LIN {X 0,Y 572.99,Z 934.788,A -85,B 0,C 180,E1 -2246.836,E2 -2246.836} C_VEL
LIN {X 0,Y 572.937,Z 937.681,A -85,B 0,C 180,E1 -2247.891,E2 -2247.891} C_VEL
LIN {X 0,Y 572.945,Z 938.936,A -85,B 0,C 180,E1 -2248.594,E2 -2248.594} C_VEL
LIN {X 0,Y 572.938,Z 939.711,A -85,B 0,C 180,E1 -2249.297,E2 -2249.297} C_VEL
LIN {X 0,Y 572.935,Z 940,A -85,B 0,C 180,E1 -2250,E2 -2250} C_VEL
LIN {X 0,Y 572.938,Z 939.711,A -85,B 0,C 180,E1 -2250.703,E2 -2250.703} C_VEL
LIN {X 0,Y 572.945,Z 938.936,A -85,B 0,C 180,E1 -2251.406,E2 -2251.406} C_VEL
LIN {X 0,Y 572.937,Z 937.68,A -85,B 0,C 180,E1 -2252.109,E2 -2252.109} C_VEL
LIN {X 0,Y 572.99,Z 934.788,A -85,B 0,C 180,E1 -2253.164,E2 -2253.164} C_VEL
LIN {X 0,Y 573.036,Z 932.147,A -85,B 0,C 180,E1 -2253.868,E2 -2253.868} C_VEL
LIN {X 0,Y 572.995,Z 926.985,A -85,B 0,C 180,E1 -2254.925,E2 -2254.925} C_VEL
LIN {X 0,Y 573.137,Z 920.188,A -85,B 0,C 180,E1 -2255.983,E2 -2255.983} C_VEL
LIN {X 0,Y 573.164,Z 912.803,A -85,B 0,C 180,E1 -2256.86,E2 -2256.86} C_VEL
LIN {X 0,Y 573.216,Z 905.405,A -85,B 0,C 180,E1 -2257.574,E2 -2257.574} C_VEL
LIN {X 0,Y 573.284,Z 897.548,A -85,B 0,C 180,E1 -2258.193,E2 -2258.193} C_VEL
LIN {X 0,Y 573.4,Z 887.734,A -85,B 0,C 180,E1 -2258.813,E2 -2258.813} C_VEL
LIN {X 0,Y 573.443,Z 876.299,A -85,B 0,C 180,E1 -2259.346,E2 -2259.346} C_VEL
LIN {X 0,Y 573.53,Z 866.245,A -85,B 0,C 180,E1 -2259.678,E2 -2259.678} C_VEL
LIN {X 0,Y 573.574,Z 857.443,A -85,B 0,C 180,E1 -2259.877,E2 -2259.877} C_VEL
LIN {X 0,Y 573.574,Z 783.105,A -85,B 0,C 180,E1 -2260.826,E2 -2260.826} C_VEL
LIN {X 0,Y 573.197,Z 780.107,A -85,B 0,C 180,E1 -2260.899,E2 -2260.899} C_VEL
LIN {X 0,Y 573.231,Z 774.077,A -85,B 0,C 180,E1 -2261.851,E2 -2261.851} C_VEL
LIN {X 0,Y 573.374,Z 755.693,A -85,B 0,C 180,E1 -2264.916,E2 -2264.916} C_VEL
LIN {X 0,Y 573.523,Z 738.39,A -85,B 0,C 180,E1 -2267.84,E2 -2267.84} C_VEL
LIN {X 0,Y 573.707,Z 721.087,A -85,B 0,C 180,E1 -2270.809,E2 -2270.809} C_VEL
LIN {X 0,Y 573.325,Z 716.043,A -85,B 0,C 180,E1 -2271.719,E2 -2271.719} C_VEL
LIN {X 0,Y 573.27,Z 715.887,A -85,B 0,C 180,E1 -2274.879,E2 -2274.879} C_VEL
LIN {X 0,Y 573.273,Z 715.885,A -85,B 0,C 180,E1 -2277.766,E2 -2277.766} C_VEL
LIN {X 0,Y 573.251,Z 715.882,A -85,B 0,C 180,E1 -2280.176,E2 -2280.176} C_VEL
LIN {X 0,Y 573.257,Z 715.884,A -85,B 0,C 180,E1 -2282.645,E2 -2282.645} C_VEL
LIN {X 0,Y 573.271,Z 715.889,A -85,B 0,C 180,E1 -2285.183,E2 -2285.183} C_VEL
LIN {X 0,Y 573.238,Z 715.891,A -85,B 0,C 180,E1 -2287.807,E2 -2287.807} C_VEL
LIN {X 0,Y 573.271,Z 715.88,A -85,B 0,C 180,E1 -2290.528,E2 -2290.528} C_VEL
LIN {X 0,Y 573.245,Z 715.894,A -85,B 0,C 180,E1 -2293.669,E2 -2293.669} C_VEL
LIN {X 0,Y 573.242,Z 715.885,A -85,B 0,C 180,E1 -2296.641,E2 -2296.641} C_VEL
LIN {X 0,Y 573.276,Z 715.885,A -85,B 0,C 180,E1 -2299.478,E2 -2299.478} C_VEL
LIN {X 0,Y 573.239,Z 715.886,A -85,B 0,C 180,E1 -2302.193,E2 -2302.193} C_VEL
LIN {X 0,Y 573.271,Z 715.881,A -85,B 0,C 180,E1 -2304.817,E2 -2304.817} C_VEL
LIN {X 0,Y 573.257,Z 715.887,A -85,B 0,C 180,E1 -2307.355,E2 -2307.355} C_VEL
LIN {X 0,Y 573.252,Z 715.893,A -85,B 0,C 180,E1 -2309.824,E2 -2309.824} C_VEL
LIN {X 0,Y 573.275,Z 715.887,A -85,B 0,C 180,E1 -2312.234,E2 -2312.234} C_VEL
LIN {X 0,Y 573.269,Z 715.882,A -85,B 0,C 180,E1 -2315.122,E2 -2315.122} C_VEL
LIN {X 0,Y 573.239,Z 715.889,A -85,B 0,C 180,E1 -2317.662,E2 -2317.662} C_VEL
LIN {X 0,Y 573.281,Z 715.882,A -85,B 0,C 180,E1 -2320.728,E2 -2320.728} C_VEL
LIN {X 0,Y 573.255,Z 715.886,A -85,B 0,C 180,E1 -2323.622,E2 -2323.622} C_VEL
LIN {X 0,Y 573.276,Z 715.884,A -85,B 0,C 180,E1 -2325.807,E2 -2325.807} C_VEL
LIN {X 0,Y 573.265,Z 715.884,A -85,B 0,C 180,E1 -2328.745,E2 -2328.745} C_VEL
LIN {X 0,Y 573.292,Z 715.88,A -85,B 0,C 180,E1 -2331.541,E2 -2331.541} C_VEL
LIN {X 0,Y 573.288,Z 715.89,A -85,B 0,C 180,E1 -2334.372,E2 -2334.372} C_VEL
LIN {X 0,Y 573.312,Z 715.875,A -85,B 0,C 180,E1 -2337.893,E2 -2337.893} C_VEL
LIN {X 0,Y 573.335,Z 715.881,A -85,B 0,C 180,E1 -2340.702,E2 -2340.702} C_VEL
LIN {X 0,Y 573.311,Z 715.883,A -85,B 0,C 180,E1 -2342.811,E2 -2342.811} C_VEL
LIN {X 0,Y 573.296,Z 715.877,A -85,B 0,C 180,E1 -2345.628,E2 -2345.628} C_VEL
LIN {X 0,Y 573.288,Z 715.883,A -85,B 0,C 180,E1 -2348.46,E2 -2348.46} C_VEL
LIN {X 0,Y 573.275,Z 715.884,A -85,B 0,C 180,E1 -2351.312,E2 -2351.312} C_VEL
LIN {X 0,Y 573.284,Z 715.884,A -85,B 0,C 180,E1 -2354.424,E2 -2354.424} C_VEL
LIN {X 0,Y 573.261,Z 715.887,A -85,B 0,C 180,E1 -2357.112,E2 -2357.112} C_VEL
LIN {X 0,Y 573.245,Z 715.885,A -85,B 0,C 180,E1 -2360.077,E2 -2360.077} C_VEL
LIN {X 0,Y 573.236,Z 715.888,A -85,B 0,C 180,E1 -2362.338,E2 -2362.338} C_VEL
LIN {X 0,Y 573.249,Z 715.885,A -85,B 0,C 180,E1 -2364.385,E2 -2364.385} C_VEL
LIN {X 0,Y 572.625,Z 715.972,A -85,B 0,C 180,E1 -2364.972,E2 -2364.972} C_VEL
LIN {X 0,Y 569.784,Z 716.327,A -85,B 0,C 180,E1 -2365.923,E2 -2365.923} C_VEL
LIN {X 0,Y 567.352,Z 716.63,A -85,B 0,C 180,E1 -2366.689,E2 -2366.689} C_VEL
LIN {X 0,Y 566.296,Z 716.757,A -85,B 0,C 180,E1 -2367.28,E2 -2367.28} C_VEL
LIN {X 0,Y 566.206,Z 716.765,A -85,B 0,C 180,E1 -2367.48,E2 -2367.48} C_VEL
LIN {X 0,Y 566.199,Z 716.764,A -85,B 0,C 180,E1 -2369.769,E2 -2369.769} C_VEL
LIN {X 0,Y 566.206,Z 716.762,A -85,B 0,C 180,E1 -2372.43,E2 -2372.43} C_VEL
LIN {X 0,Y 566.182,Z 716.77,A -85,B 0,C 180,E1 -2374.989,E2 -2374.989} C_VEL
LIN {X 0,Y 566.197,Z 716.77,A -85,B 0,C 180,E1 -2377.461,E2 -2377.461} C_VEL
LIN {X 0,Y 566.208,Z 716.759,A -85,B 0,C 180,E1 -2380.199,E2 -2380.199} C_VEL
LIN {X 0,Y 566.202,Z 716.759,A -85,B 0,C 180,E1 -2383.054,E2 -2383.054} C_VEL
LIN {X 0,Y 566.195,Z 716.765,A -85,B 0,C 180,E1 -2386.049,E2 -2386.049} C_VEL
LIN {X 0,Y 566.205,Z 716.768,A -85,B 0,C 180,E1 -2389.215,E2 -2389.215} C_VEL
LIN {X 0,Y 566.186,Z 716.771,A -85,B 0,C 180,E1 -2391.637,E2 -2391.637} C_VEL
LIN {X 0,Y 566.163,Z 716.769,A -85,B 0,C 180,E1 -2394.308,E2 -2394.308} C_VEL
LIN {X 0,Y 566.2,Z 716.763,A -85,B 0,C 180,E1 -2396.896,E2 -2396.896} C_VEL
LIN {X 0,Y 566.176,Z 716.769,A -85,B 0,C 180,E1 -2399.407,E2 -2399.407} C_VEL
LIN {X 0,Y 566.188,Z 716.774,A -85,B 0,C 180,E1 -2401.856,E2 -2401.856} C_VEL
LIN {X 0,Y 566.201,Z 716.767,A -85,B 0,C 180,E1 -2404.25,E2 -2404.25} C_VEL
LIN {X 0,Y 566.169,Z 716.767,A -85,B 0,C 180,E1 -2406.72,E2 -2406.72} C_VEL
LIN {X 0,Y 566.207,Z 716.769,A -85,B 0,C 180,E1 -2409.663,E2 -2409.663} C_VEL
LIN {X 0,Y 566.246,Z 716.863,A -85,B 0,C 180,E1 -2411.736,E2 -2411.736} C_VEL
LIN {X 0,Y 566.229,Z 726.34,A -85,B 0,C 180,E1 -2413.783,E2 -2413.783} C_VEL
LIN {X 0,Y 566.15,Z 738.526,A -85,B 0,C 180,E1 -2416.358,E2 -2416.358} C_VEL
LIN {X 0,Y 566.101,Z 751.445,A -85,B 0,C 180,E1 -2419.016,E2 -2419.016} C_VEL
LIN {X 0,Y 566.291,Z 753.402,A -85,B 0,C 180,E1 -2419.081,E2 -2419.081} C_VEL
LIN {X 0,Y 566.703,Z 760.329,A -85,B 0,C 180,E1 -2419.177,E2 -2419.177} C_VEL
LIN {X 0,Y 566.574,Z 826.154,A -85,B 0,C 180,E1 -2420.022,E2 -2420.022} C_VEL
LIN {X 0,Y 566.563,Z 835.43,A -85,B 0,C 180,E1 -2420.224,E2 -2420.224} C_VEL
LIN {X 0,Y 566.459,Z 845.107,A -85,B 0,C 180,E1 -2420.538,E2 -2420.538} C_VEL
LIN {X 0,Y 566.383,Z 855.187,A -85,B 0,C 180,E1 -2420.987,E2 -2420.987} C_VEL
LIN {X 0,Y 566.293,Z 865.698,A -85,B 0,C 180,E1 -2421.615,E2 -2421.615} C_VEL
LIN {X 0,Y 566.171,Z 873.875,A -85,B 0,C 180,E1 -2422.242,E2 -2422.242} C_VEL
LIN {X 0,Y 566.097,Z 881.688,A -85,B 0,C 180,E1 -2422.981,E2 -2422.981} C_VEL
LIN {X 0,Y 566.087,Z 888.422,A -85,B 0,C 180,E1 -2423.764,E2 -2423.764} C_VEL
LIN {X 0,Y 565.946,Z 894.663,A -85,B 0,C 180,E1 -2424.656,E2 -2424.656} C_VEL
LIN {X 0,Y 565.96,Z 900.44,A -85,B 0,C 180,E1 -2425.727,E2 -2425.727} C_VEL
LIN {X 0,Y 565.913,Z 904.644,A -85,B 0,C 180,E1 -2426.796,E2 -2426.796} C_VEL
LIN {X 0,Y 565.841,Z 907.582,A -85,B 0,C 180,E1 -2427.865,E2 -2427.865} C_VEL
LIN {X 0,Y 565.843,Z 908.875,A -85,B 0,C 180,E1 -2428.577,E2 -2428.577} C_VEL
LIN {X 0,Y 565.837,Z 909.691,A -85,B 0,C 180,E1 -2429.288,E2 -2429.288} C_VEL
LIN {X 0,Y 565.837,Z 909.996,A -85,B 0,C 180,E1 -2430,E2 -2430} C_VEL
LIN {X 0,Y 565.838,Z 909.731,A -85,B 0,C 180,E1 -2430.712,E2 -2430.712} C_VEL
LIN {X 0,Y 565.845,Z 908.997,A -85,B 0,C 180,E1 -2431.423,E2 -2431.423} C_VEL
LIN {X 0,Y 565.841,Z 907.784,A -85,B 0,C 180,E1 -2432.135,E2 -2432.135} C_VEL
LIN {X 0,Y 565.913,Z 904.935,A -85,B 0,C 180,E1 -2433.204,E2 -2433.204} C_VEL
LIN {X 0,Y 565.935,Z 902.34,A -85,B 0,C 180,E1 -2433.916,E2 -2433.916} C_VEL
LIN {X 0,Y 565.963,Z 899.141,A -85,B 0,C 180,E1 -2434.63,E2 -2434.63} C_VEL
LIN {X 0,Y 565.987,Z 894.08,A -85,B 0,C 180,E1 -2435.522,E2 -2435.522} C_VEL
LIN {X 0,Y 566.077,Z 889.136,A -85,B 0,C 180,E1 -2436.237,E2 -2436.237} C_VEL
LIN {X 0,Y 566.083,Z 883.163,A -85,B 0,C 180,E1 -2436.954,E2 -2436.954} C_VEL
LIN {X 0,Y 566.166,Z 874.9,A -85,B 0,C 180,E1 -2437.758,E2 -2437.758} C_VEL
LIN {X 0,Y 566.265,Z 866.932,A -85,B 0,C 180,E1 -2438.385,E2 -2438.385} C_VEL
LIN {X 0,Y 566.374,Z 856.952,A -85,B 0,C 180,E1 -2439.013,E2 -2439.013} C_VEL
LIN {X 0,Y 566.445,Z 846.308,A -85,B 0,C 180,E1 -2439.507,E2 -2439.507} C_VEL
LIN {X 0,Y 566.527,Z 836.254,A -85,B 0,C 180,E1 -2439.844,E2 -2439.844} C_VEL
LIN {X 0,Y 566.597,Z 827.442,A -85,B 0,C 180,E1 -2440.045,E2 -2440.045} C_VEL
LIN {X 0,Y 566.693,Z 756.444,A -85,B 0,C 180,E1 -2440.962,E2 -2440.962} C_VEL
LIN {X 0,Y 566.121,Z 751.723,A -85,B 0,C 180,E1 -2441.058,E2 -2441.058} C_VEL
LIN {X 0,Y 566.068,Z 750.455,A -85,B 0,C 180,E1 -2441.239,E2 -2441.239} C_VEL
LIN {X 0,Y 566.204,Z 734.904,A -85,B 0,C 180,E1 -2444.494,E2 -2444.494} C_VEL
LIN {X 0,Y 566.307,Z 719.797,A -85,B 0,C 180,E1 -2447.701,E2 -2447.701} C_VEL
LIN {X 0,Y 566.278,Z 716.86,A -85,B 0,C 180,E1 -2448.356,E2 -2448.356} C_VEL
LIN {X 0,Y 566.21,Z 716.763,A -85,B 0,C 180,E1 -2451.42,E2 -2451.42} C_VEL
LIN {X 0,Y 566.179,Z 716.775,A -85,B 0,C 180,E1 -2454.182,E2 -2454.182} C_VEL
LIN {X 0,Y 566.173,Z 716.771,A -85,B 0,C 180,E1 -2456.652,E2 -2456.652} C_VEL
LIN {X 0,Y 566.2,Z 716.764,A -85,B 0,C 180,E1 -2459.671,E2 -2459.671} C_VEL
LIN {X 0,Y 566.204,Z 716.771,A -85,B 0,C 180,E1 -2462.43,E2 -2462.43} C_VEL
LIN {X 0,Y 566.179,Z 716.768,A -85,B 0,C 180,E1 -2464.989,E2 -2464.989} C_VEL
LIN {X 0,Y 566.197,Z 716.761,A -85,B 0,C 180,E1 -2467.461,E2 -2467.461} C_VEL
LIN {X 0,Y 566.208,Z 716.764,A -85,B 0,C 180,E1 -2470.199,E2 -2470.199} C_VEL
LIN {X 0,Y 566.202,Z 716.766,A -85,B 0,C 180,E1 -2473.054,E2 -2473.054} C_VEL
LIN {X 0,Y 566.195,Z 716.762,A -85,B 0,C 180,E1 -2476.049,E2 -2476.049} C_VEL
LIN {X 0,Y 566.205,Z 716.762,A -85,B 0,C 180,E1 -2479.215,E2 -2479.215} C_VEL
LIN {X 0,Y 566.182,Z 716.765,A -85,B 0,C 180,E1 -2481.636,E2 -2481.636} C_VEL
LIN {X 0,Y 566.164,Z 716.77,A -85,B 0,C 180,E1 -2484.308,E2 -2484.308} C_VEL
LIN {X 0,Y 566.206,Z 716.77,A -85,B 0,C 180,E1 -2486.897,E2 -2486.897} C_VEL
LIN {X 0,Y 566.176,Z 716.769,A -85,B 0,C 180,E1 -2489.407,E2 -2489.407} C_VEL
LIN {X 0,Y 566.214,Z 716.761,A -85,B 0,C 180,E1 -2491.857,E2 -2491.857} C_VEL
LIN {X 0,Y 566.209,Z 716.759,A -85,B 0,C 180,E1 -2494.251,E2 -2494.251} C_VEL
LIN {X 0,Y 566.171,Z 716.77,A -85,B 0,C 180,E1 -2496.719,E2 -2496.719} C_VEL
LIN {X 0,Y 566.211,Z 716.763,A -85,B 0,C 180,E1 -2499.663,E2 -2499.663} C_VEL
LIN {X 0,Y 566.202,Z 716.762,A -85,B 0,C 180,E1 -2502.668,E2 -2502.668} C_VEL
LIN {X 0,Y 566.237,Z 716.762,A -85,B 0,C 180,E1 -2505.627,E2 -2505.627} C_VEL
LIN {X 0,Y 566.238,Z 716.76,A -85,B 0,C 180,E1 -2508.675,E2 -2508.675} C_VEL
LIN {X 0,Y 566.231,Z 716.764,A -85,B 0,C 180,E1 -2511.434,E2 -2511.434} C_VEL
LIN {X 0,Y 566.264,Z 716.753,A -85,B 0,C 180,E1 -2514.302,E2 -2514.302} C_VEL
LIN {X 0,Y 566.286,Z 716.756,A -85,B 0,C 180,E1 -2517.866,E2 -2517.866} C_VEL
LIN {X 0,Y 566.305,Z 716.748,A -85,B 0,C 180,E1 -2520.711,E2 -2520.711} C_VEL
LIN {X 0,Y 566.277,Z 716.75,A -85,B 0,C 180,E1 -2522.845,E2 -2522.845} C_VEL
LIN {X 0,Y 566.256,Z 716.766,A -85,B 0,C 180,E1 -2525.698,E2 -2525.698} C_VEL
LIN {X 0,Y 566.236,Z 716.758,A -85,B 0,C 180,E1 -2528.566,E2 -2528.566} C_VEL
LIN {X 0,Y 566.244,Z 716.761,A -85,B 0,C 180,E1 -2531.454,E2 -2531.454} C_VEL
LIN {X 0,Y 566.237,Z 716.758,A -85,B 0,C 180,E1 -2534.507,E2 -2534.507} C_VEL
LIN {X 0,Y 566.206,Z 716.764,A -85,B 0,C 180,E1 -2537.331,E2 -2537.331} C_VEL
LIN {X 0,Y 566.216,Z 716.762,A -85,B 0,C 180,E1 -2540.337,E2 -2540.337} C_VEL
LIN {X 0,Y 566.192,Z 716.764,A -85,B 0,C 180,E1 -2543.404,E2 -2543.404} C_VEL
LIN {X 0,Y 566.215,Z 716.767,A -85,B 0,C 180,E1 -2545.749,E2 -2545.749} C_VEL
LIN {X 0,Y 566.208,Z 716.768,A -85,B 0,C 180,E1 -2548.203,E2 -2548.203} C_VEL
LIN {X 0,Y 566.201,Z 716.762,A -85,B 0,C 180,E1 -2551.078,E2 -2551.078} C_VEL
LIN {X 0,Y 566.214,Z 716.764,A -85,B 0,C 180,E1 -2553.734,E2 -2553.734} C_VEL
LIN {X 0,Y 566.218,Z 716.762,A -85,B 0,C 180,E1 -2556.568,E2 -2556.568} C_VEL
LIN {X 0,Y 566.214,Z 716.754,A -85,B 0,C 180,E1 -2559.686,E2 -2559.686} C_VEL
LIN {X 0,Y 566.215,Z 716.763,A -85,B 0,C 180,E1 -2562.087,E2 -2562.087} C_VEL
LIN {X 0,Y 566.174,Z 716.768,A -85,B 0,C 180,E1 -2565.036,E2 -2565.036} C_VEL
LIN {X 0,Y 566.22,Z 716.763,A -85,B 0,C 180,E1 -2568.136,E2 -2568.136} C_VEL
LIN {X 0,Y 566.223,Z 716.767,A -85,B 0,C 180,E1 -2570.727,E2 -2570.727} C_VEL
LIN {X 0,Y 566.219,Z 716.76,A -85,B 0,C 180,E1 -2573.783,E2 -2573.783} C_VEL
LIN {X 0,Y 566.214,Z 716.766,A -85,B 0,C 180,E1 -2576.266,E2 -2576.266} C_VEL
LIN {X 0,Y 566.2,Z 716.766,A -85,B 0,C 180,E1 -2578.922,E2 -2578.922} C_VEL
LIN {X 0,Y 566.212,Z 716.762,A -85,B 0,C 180,E1 -2581.857,E2 -2581.857} C_VEL
LIN {X 0,Y 566.217,Z 716.763,A -85,B 0,C 180,E1 -2584.251,E2 -2584.251} C_VEL
LIN {X 0,Y 566.174,Z 716.774,A -85,B 0,C 180,E1 -2586.718,E2 -2586.718} C_VEL
LIN {X 0,Y 566.272,Z 716.893,A -85,B 0,C 180,E1 -2588.141,E2 -2588.141} C_VEL
LIN {X 0,Y 566.724,Z 721.087,A -85,B 0,C 180,E1 -2588.922,E2 -2588.922} C_VEL
LIN {X 0,Y 566.56,Z 736.227,A -85,B 0,C 180,E1 -2591.559,E2 -2591.559} C_VEL
LIN {X 0,Y 566.379,Z 752.448,A -85,B 0,C 180,E1 -2594.342,E2 -2594.342} C_VEL
LIN {X 0,Y 566.207,Z 768.67,A -85,B 0,C 180,E1 -2597.09,E2 -2597.09} C_VEL
LIN {X 0,Y 566.127,Z 779.977,A -85,B 0,C 180,E1 -2598.952,E2 -2598.952} C_VEL
LIN {X 0,Y 566.413,Z 782.311,A -85,B 0,C 180,E1 -2599.025,E2 -2599.025} C_VEL
LIN {X 0,Y 566.687,Z 793.79,A -85,B 0,C 180,E1 -2599.175,E2 -2599.175} C_VEL
LIN {X 0,Y 566.582,Z 857.436,A -85,B 0,C 180,E1 -2599.999,E2 -2599.999} C_VEL
LIN {X 0,Y 566.556,Z 867.073,A -85,B 0,C 180,E1 -2600.224,E2 -2600.224} C_VEL
LIN {X 0,Y 566.452,Z 878.612,A -85,B 0,C 180,E1 -2600.628,E2 -2600.628} C_VEL
LIN {X 0,Y 566.332,Z 889.232,A -85,B 0,C 180,E1 -2601.166,E2 -2601.166} C_VEL
LIN {X 0,Y 566.239,Z 897.544,A -85,B 0,C 180,E1 -2601.704,E2 -2601.704} C_VEL
LIN {X 0,Y 566.168,Z 905.403,A -85,B 0,C 180,E1 -2602.331,E2 -2602.331} C_VEL
LIN {X 0,Y 566.088,Z 913.228,A -85,B 0,C 180,E1 -2603.099,E2 -2603.099} C_VEL
LIN {X 0,Y 566.057,Z 921.433,A -85,B 0,C 180,E1 -2604.121,E2 -2604.121} C_VEL
LIN {X 0,Y 565.906,Z 926.987,A -85,B 0,C 180,E1 -2605.013,E2 -2605.013} C_VEL
LIN {X 0,Y 565.943,Z 932.148,A -85,B 0,C 180,E1 -2606.084,E2 -2606.084} C_VEL
LIN {X 0,Y 565.912,Z 934.789,A -85,B 0,C 180,E1 -2606.796,E2 -2606.796} C_VEL
LIN {X 0,Y 565.838,Z 937.681,A -85,B 0,C 180,E1 -2607.865,E2 -2607.865} C_VEL
LIN {X 0,Y 565.844,Z 938.936,A -85,B 0,C 180,E1 -2608.577,E2 -2608.577} C_VEL
LIN {X 0,Y 565.839,Z 939.711,A -85,B 0,C 180,E1 -2609.288,E2 -2609.288} C_VEL
LIN {X 0,Y 565.836,Z 940,A -85,B 0,C 180,E1 -2610,E2 -2610} C_VEL
LIN {X 0,Y 565.839,Z 939.711,A -85,B 0,C 180,E1 -2610.712,E2 -2610.712} C_VEL
LIN {X 0,Y 565.844,Z 938.936,A -85,B 0,C 180,E1 -2611.423,E2 -2611.423} C_VEL
LIN {X 0,Y 565.838,Z 937.681,A -85,B 0,C 180,E1 -2612.135,E2 -2612.135} C_VEL
LIN {X 0,Y 565.912,Z 934.788,A -85,B 0,C 180,E1 -2613.204,E2 -2613.204} C_VEL
LIN {X 0,Y 565.943,Z 932.148,A -85,B 0,C 180,E1 -2613.916,E2 -2613.916} C_VEL
LIN {X 0,Y 565.906,Z 926.985,A -85,B 0,C 180,E1 -2614.987,E2 -2614.987} C_VEL
LIN {X 0,Y 566.082,Z 920.187,A -85,B 0,C 180,E1 -2616.058,E2 -2616.058} C_VEL
LIN {X 0,Y 566.091,Z 913.178,A -85,B 0,C 180,E1 -2616.907,E2 -2616.907} C_VEL
LIN {X 0,Y 566.168,Z 905.406,A -85,B 0,C 180,E1 -2617.669,E2 -2617.669} C_VEL
LIN {X 0,Y 566.239,Z 897.546,A -85,B 0,C 180,E1 -2618.296,E2 -2618.296} C_VEL
LIN {X 0,Y 566.378,Z 887.732,A -85,B 0,C 180,E1 -2618.923,E2 -2618.923} C_VEL
LIN {X 0,Y 566.448,Z 876.301,A -85,B 0,C 180,E1 -2619.462,E2 -2619.462} C_VEL
LIN {X 0,Y 566.537,Z 866.245,A -85,B 0,C 180,E1 -2619.799,E2 -2619.799} C_VEL
LIN {X 0,Y 566.582,Z 857.442,A -85,B 0,C 180,E1 -2620.001,E2 -2620.001} C_VEL
LIN {X 0,Y 566.698,Z 787.78,A -85,B 0,C 180,E1 -2620.9,E2 -2620.9} C_VEL
LIN {X 0,Y 566.396,Z 782.296,A -85,B 0,C 180,E1 -2620.976,E2 -2620.976} C_VEL
LIN {X 0,Y 566.138,Z 779.979,A -85,B 0,C 180,E1 -2621.047,E2 -2621.047} C_VEL
LIN {X 0,Y 566.269,Z 764.344,A -85,B 0,C 180,E1 -2623.639,E2 -2623.639} C_VEL
LIN {X 0,Y 566.437,Z 747.041,A -85,B 0,C 180,E1 -2626.581,E2 -2626.581} C_VEL
LIN {X 0,Y 566.611,Z 732.105,A -85,B 0,C 180,E1 -2629.154,E2 -2629.154} C_VEL
LIN {X 0,Y 566.694,Z 719.879,A -85,B 0,C 180,E1 -2631.292,E2 -2631.292} C_VEL
LIN {X 0,Y 566.254,Z 716.808,A -85,B 0,C 180,E1 -2631.896,E2 -2631.896} C_VEL
LIN {X 0,Y 566.219,Z 716.768,A -85,B 0,C 180,E1 -2635.03,E2 -2635.03} C_VEL
LIN {X 0,Y 566.213,Z 716.771,A -85,B 0,C 180,E1 -2637.339,E2 -2637.339} C_VEL
LIN {X 0,Y 566.204,Z 716.763,A -85,B 0,C 180,E1 -2639.769,E2 -2639.769} C_VEL
LIN {X 0,Y 566.209,Z 716.761,A -85,B 0,C 180,E1 -2642.431,E2 -2642.431} C_VEL
LIN {X 0,Y 566.216,Z 716.765,A -85,B 0,C 180,E1 -2644.995,E2 -2644.995} C_VEL
LIN {X 0,Y 566.198,Z 716.774,A -85,B 0,C 180,E1 -2647.461,E2 -2647.461} C_VEL
LIN {X 0,Y 566.229,Z 716.758,A -85,B 0,C 180,E1 -2650.197,E2 -2650.197} C_VEL
LIN {X 0,Y 566.202,Z 716.764,A -85,B 0,C 180,E1 -2653.054,E2 -2653.054} C_VEL
LIN {X 0,Y 566.2,Z 716.766,A -85,B 0,C 180,E1 -2656.049,E2 -2656.049} C_VEL
LIN {X 0,Y 566.213,Z 716.758,A -85,B 0,C 180,E1 -2658.864,E2 -2658.864} C_VEL
LIN {X 0,Y 566.192,Z 716.764,A -85,B 0,C 180,E1 -2661.637,E2 -2661.637} C_VEL
LIN {X 0,Y 566.215,Z 716.763,A -85,B 0,C 180,E1 -2664.312,E2 -2664.312} C_VEL
LIN {X 0,Y 566.231,Z 716.759,A -85,B 0,C 180,E1 -2666.899,E2 -2666.899} C_VEL
LIN {X 0,Y 566.19,Z 716.766,A -85,B 0,C 180,E1 -2669.408,E2 -2669.408} C_VEL
LIN {X 0,Y 566.231,Z 716.766,A -85,B 0,C 180,E1 -2671.858,E2 -2671.858} C_VEL
LIN {X 0,Y 566.215,Z 716.767,A -85,B 0,C 180,E1 -2674.251,E2 -2674.251} C_VEL
LIN {X 0,Y 566.194,Z 716.763,A -85,B 0,C 180,E1 -2676.714,E2 -2676.714} C_VEL
LIN {X 0,Y 566.216,Z 716.761,A -85,B 0,C 180,E1 -2679.663,E2 -2679.663} C_VEL
LIN {X 0,Y 566.206,Z 716.765,A -85,B 0,C 180,E1 -2682.669,E2 -2682.669} C_VEL
LIN {X 0,Y 566.237,Z 716.759,A -85,B 0,C 180,E1 -2685.627,E2 -2685.627} C_VEL
LIN {X 0,Y 566.237,Z 716.76,A -85,B 0,C 180,E1 -2688.675,E2 -2688.675} C_VEL
LIN {X 0,Y 566.235,Z 716.758,A -85,B 0,C 180,E1 -2691.434,E2 -2691.434} C_VEL
LIN {X 0,Y 566.257,Z 716.765,A -85,B 0,C 180,E1 -2694.302,E2 -2694.302} C_VEL
LIN {X 0,Y 566.283,Z 716.75,A -85,B 0,C 180,E1 -2697.866,E2 -2697.866} C_VEL
LIN {X 0,Y 566.305,Z 716.757,A -85,B 0,C 180,E1 -2700.711,E2 -2700.711} C_VEL
LIN {X 0,Y 566.277,Z 716.759,A -85,B 0,C 180,E1 -2702.846,E2 -2702.846} C_VEL
LIN {X 0,Y 566.265,Z 716.753,A -85,B 0,C 180,E1 -2705.698,E2 -2705.698} C_VEL
LIN {X 0,Y 566.231,Z 716.763,A -85,B 0,C 180,E1 -2708.566,E2 -2708.566} C_VEL
LIN {X 0,Y 566.244,Z 716.758,A -85,B 0,C 180,E1 -2711.454,E2 -2711.454} C_VEL
LIN {X 0,Y 566.237,Z 716.763,A -85,B 0,C 180,E1 -2714.507,E2 -2714.507} C_VEL
LIN {X 0,Y 566.201,Z 716.763,A -85,B 0,C 180,E1 -2717.332,E2 -2717.332} C_VEL
LIN {X 0,Y 566.211,Z 716.763,A -85,B 0,C 180,E1 -2720.337,E2 -2720.337} C_VEL
LIN {X 0,Y 566.171,Z 716.771,A -85,B 0,C 180,E1 -2723.281,E2 -2723.281} C_VEL
LIN {X 0,Y 566.21,Z 716.759,A -85,B 0,C 180,E1 -2725.749,E2 -2725.749} C_VEL
LIN {X 0,Y 566.206,Z 716.765,A -85,B 0,C 180,E1 -2727.48,E2 -2727.48} C_VEL
LIN {X 0,Y 565.525,Z 716.849,A -85,B 0,C 180,E1 -2728.074,E2 -2728.074} C_VEL
LIN {X 0,Y 562.657,Z 717.213,A -85,B 0,C 180,E1 -2729.037,E2 -2729.037} C_VEL
LIN {X 0,Y 560.246,Z 717.508,A -85,B 0,C 180,E1 -2729.813,E2 -2729.813} C_VEL
LIN {X 0,Y 559.218,Z 717.634,A -85,B 0,C 180,E1 -2730.412,E2 -2730.412} C_VEL
LIN {X 0,Y 559.138,Z 717.645,A -85,B 0,C 180,E1 -2730.614,E2 -2730.614} C_VEL
LIN {X 0,Y 559.155,Z 717.642,A -85,B 0,C 180,E1 -2732.715,E2 -2732.715} C_VEL
LIN {X 0,Y 559.129,Z 717.653,A -85,B 0,C 180,E1 -2735.324,E2 -2735.324} C_VEL
LIN {X 0,Y 559.131,Z 717.644,A -85,B 0,C 180,E1 -2738.018,E2 -2738.018} C_VEL
LIN {X 0,Y 559.157,Z 717.639,A -85,B 0,C 180,E1 -2740.813,E2 -2740.813} C_VEL
LIN {X 0,Y 559.139,Z 717.644,A -85,B 0,C 180,E1 -2743.734,E2 -2743.734} C_VEL
LIN {X 0,Y 559.147,Z 717.643,A -85,B 0,C 180,E1 -2746.804,E2 -2746.804} C_VEL
LIN {X 0,Y 559.156,Z 717.645,A -85,B 0,C 180,E1 -2749.188,E2 -2749.188} C_VEL
LIN {X 0,Y 559.133,Z 717.645,A -85,B 0,C 180,E1 -2751.982,E2 -2751.982} C_VEL
LIN {X 0,Y 559.132,Z 717.644,A -85,B 0,C 180,E1 -2754.787,E2 -2754.787} C_VEL
LIN {X 0,Y 559.154,Z 717.646,A -85,B 0,C 180,E1 -2757.365,E2 -2757.365} C_VEL
LIN {X 0,Y 559.146,Z 717.646,A -85,B 0,C 180,E1 -2760.143,E2 -2760.143} C_VEL
LIN {X 0,Y 559.161,Z 717.642,A -85,B 0,C 180,E1 -2763.175,E2 -2763.175} C_VEL
LIN {X 0,Y 559.13,Z 717.649,A -85,B 0,C 180,E1 -2765.494,E2 -2765.494} C_VEL
LIN {X 0,Y 559.173,Z 717.64,A -85,B 0,C 180,E1 -2768.624,E2 -2768.624} C_VEL
LIN {X 0,Y 559.225,Z 717.744,A -85,B 0,C 180,E1 -2771.688,E2 -2771.688} C_VEL
LIN {X 0,Y 559.227,Z 726.343,A -85,B 0,C 180,E1 -2773.575,E2 -2773.575} C_VEL
LIN {X 0,Y 559.098,Z 740.27,A -85,B 0,C 180,E1 -2776.553,E2 -2776.553} C_VEL
LIN {X 0,Y 559.034,Z 751.587,A -85,B 0,C 180,E1 -2778.914,E2 -2778.914} C_VEL
LIN {X 0,Y 559.716,Z 759.135,A -85,B 0,C 180,E1 -2779.024,E2 -2779.024} C_VEL
LIN {X 0,Y 559.585,Z 826.187,A -85,B 0,C 180,E1 -2779.896,E2 -2779.896} C_VEL
LIN {X 0,Y 559.557,Z 835.45,A -85,B 0,C 180,E1 -2780.101,E2 -2780.101} C_VEL
LIN {X 0,Y 559.474,Z 845.125,A -85,B 0,C 180,E1 -2780.419,E2 -2780.419} C_VEL
LIN {X 0,Y 559.358,Z 855.202,A -85,B 0,C 180,E1 -2780.873,E2 -2780.873} C_VEL
LIN {X 0,Y 559.258,Z 865.703,A -85,B 0,C 180,E1 -2781.509,E2 -2781.509} C_VEL
LIN {X 0,Y 559.135,Z 873.879,A -85,B 0,C 180,E1 -2782.143,E2 -2782.143} C_VEL
LIN {X 0,Y 559.058,Z 880.622,A -85,B 0,C 180,E1 -2782.778,E2 -2782.778} C_VEL
LIN {X 0,Y 558.986,Z 887.005,A -85,B 0,C 180,E1 -2783.503,E2 -2783.503} C_VEL
LIN {X 0,Y 558.969,Z 892.317,A -85,B 0,C 180,E1 -2784.227,E2 -2784.227} C_VEL
LIN {X 0,Y 558.832,Z 896.749,A -85,B 0,C 180,E1 -2784.95,E2 -2784.95} C_VEL
LIN {X 0,Y 558.893,Z 900.443,A -85,B 0,C 180,E1 -2785.673,E2 -2785.673} C_VEL
LIN {X 0,Y 558.837,Z 904.646,A -85,B 0,C 180,E1 -2786.756,E2 -2786.756} C_VEL
LIN {X 0,Y 558.747,Z 907.584,A -85,B 0,C 180,E1 -2787.837,E2 -2787.837} C_VEL
LIN {X 0,Y 558.743,Z 908.875,A -85,B 0,C 180,E1 -2788.558,E2 -2788.558} C_VEL
LIN {X 0,Y 558.737,Z 909.691,A -85,B 0,C 180,E1 -2789.279,E2 -2789.279} C_VEL
LIN {X 0,Y 558.738,Z 909.996,A -85,B 0,C 180,E1 -2790,E2 -2790} C_VEL
LIN {X 0,Y 558.738,Z 909.73,A -85,B 0,C 180,E1 -2790.721,E2 -2790.721} C_VEL
LIN {X 0,Y 558.745,Z 908.995,A -85,B 0,C 180,E1 -2791.442,E2 -2791.442} C_VEL
LIN {X 0,Y 558.747,Z 907.784,A -85,B 0,C 180,E1 -2792.163,E2 -2792.163} C_VEL
LIN {X 0,Y 558.836,Z 904.934,A -85,B 0,C 180,E1 -2793.244,E2 -2793.244} C_VEL
LIN {X 0,Y 558.894,Z 900.821,A -85,B 0,C 180,E1 -2794.327,E2 -2794.327} C_VEL
LIN {X 0,Y 558.881,Z 895.243,A -85,B 0,C 180,E1 -2795.412,E2 -2795.412} C_VEL
LIN {X 0,Y 558.995,Z 889.131,A -85,B 0,C 180,E1 -2796.316,E2 -2796.316} C_VEL
LIN {X 0,Y 559.025,Z 883.338,A -85,B 0,C 180,E1 -2797.023,E2 -2797.023} C_VEL
LIN {X 0,Y 559.12,Z 875.911,A -85,B 0,C 180,E1 -2797.766,E2 -2797.766} C_VEL
LIN {X 0,Y 559.223,Z 868.155,A -85,B 0,C 180,E1 -2798.401,E2 -2798.401} C_VEL
LIN {X 0,Y 559.288,Z 859.973,A -85,B 0,C 180,E1 -2798.946,E2 -2798.946} C_VEL
LIN {X 0,Y 559.427,Z 849.576,A -85,B 0,C 180,E1 -2799.491,E2 -2799.491} C_VEL
LIN {X 0,Y 559.551,Z 837.896,A -85,B 0,C 180,E1 -2799.922,E2 -2799.922} C_VEL
LIN {X 0,Y 559.622,Z 827.409,A -85,B 0,C 180,E1 -2800.172,E2 -2800.172} C_VEL
LIN {X 0,Y 559.556,Z 755.577,A -85,B 0,C 180,E1 -2801.114,E2 -2801.114} C_VEL
LIN {X 0,Y 559.017,Z 751.601,A -85,B 0,C 180,E1 -2801.209,E2 -2801.209} C_VEL
LIN {X 0,Y 559.012,Z 750.878,A -85,B 0,C 180,E1 -2801.295,E2 -2801.295} C_VEL
LIN {X 0,Y 559.154,Z 735.389,A -85,B 0,C 180,E1 -2804.576,E2 -2804.576} C_VEL
LIN {X 0,Y 559.283,Z 721.536,A -85,B 0,C 180,E1 -2807.553,E2 -2807.553} C_VEL
LIN {X 0,Y 559.219,Z 717.738,A -85,B 0,C 180,E1 -2808.407,E2 -2808.407} C_VEL
LIN {X 0,Y 559.156,Z 717.643,A -85,B 0,C 180,E1 -2811.549,E2 -2811.549} C_VEL
LIN {X 0,Y 559.129,Z 717.65,A -85,B 0,C 180,E1 -2814.506,E2 -2814.506} C_VEL
LIN {X 0,Y 559.131,Z 717.645,A -85,B 0,C 180,E1 -2816.904,E2 -2816.904} C_VEL
LIN {X 0,Y 559.145,Z 717.645,A -85,B 0,C 180,E1 -2819.856,E2 -2819.856} C_VEL
LIN {X 0,Y 559.153,Z 717.646,A -85,B 0,C 180,E1 -2822.716,E2 -2822.716} C_VEL
LIN {X 0,Y 559.128,Z 717.645,A -85,B 0,C 180,E1 -2825.324,E2 -2825.324} C_VEL
LIN {X 0,Y 559.133,Z 717.644,A -85,B 0,C 180,E1 -2828.018,E2 -2828.018} C_VEL
LIN {X 0,Y 559.156,Z 717.646,A -85,B 0,C 180,E1 -2830.813,E2 -2830.813} C_VEL
LIN {X 0,Y 559.139,Z 717.643,A -85,B 0,C 180,E1 -2833.734,E2 -2833.734} C_VEL
LIN {X 0,Y 559.146,Z 717.641,A -85,B 0,C 180,E1 -2836.804,E2 -2836.804} C_VEL
LIN {X 0,Y 559.156,Z 717.64,A -85,B 0,C 180,E1 -2839.187,E2 -2839.187} C_VEL
LIN {X 0,Y 559.131,Z 717.643,A -85,B 0,C 180,E1 -2841.982,E2 -2841.982} C_VEL
LIN {X 0,Y 559.133,Z 717.653,A -85,B 0,C 180,E1 -2844.787,E2 -2844.787} C_VEL
LIN {X 0,Y 559.156,Z 717.642,A -85,B 0,C 180,E1 -2847.365,E2 -2847.365} C_VEL
LIN {X 0,Y 559.146,Z 717.642,A -85,B 0,C 180,E1 -2850.143,E2 -2850.143} C_VEL
LIN {X 0,Y 559.172,Z 717.642,A -85,B 0,C 180,E1 -2853.173,E2 -2853.173} C_VEL
LIN {X 0,Y 559.157,Z 717.642,A -85,B 0,C 180,E1 -2855.495,E2 -2855.495} C_VEL
LIN {X 0,Y 559.174,Z 717.641,A -85,B 0,C 180,E1 -2858.624,E2 -2858.624} C_VEL
LIN {X 0,Y 559.164,Z 717.645,A -85,B 0,C 180,E1 -2860.926,E2 -2860.926} C_VEL
LIN {X 0,Y 559.168,Z 717.637,A -85,B 0,C 180,E1 -2863.948,E2 -2863.948} C_VEL
LIN {X 0,Y 559.173,Z 717.638,A -85,B 0,C 180,E1 -2866.184,E2 -2866.184} C_VEL
LIN {X 0,Y 559.198,Z 717.642,A -85,B 0,C 180,E1 -2869.133,E2 -2869.133} C_VEL
LIN {X 0,Y 559.203,Z 717.63,A -85,B 0,C 180,E1 -2872.054,E2 -2872.054} C_VEL
LIN {X 0,Y 559.258,Z 717.629,A -85,B 0,C 180,E1 -2874.953,E2 -2874.953} C_VEL
LIN {X 0,Y 559.257,Z 717.632,A -85,B 0,C 180,E1 -2877.839,E2 -2877.839} C_VEL
LIN {X 0,Y 559.275,Z 717.624,A -85,B 0,C 180,E1 -2880.72,E2 -2880.72} C_VEL
LIN {X 0,Y 559.243,Z 717.626,A -85,B 0,C 180,E1 -2882.881,E2 -2882.881} C_VEL
LIN {X 0,Y 559.226,Z 717.64,A -85,B 0,C 180,E1 -2885.77,E2 -2885.77} C_VEL
LIN {X 0,Y 559.194,Z 717.635,A -85,B 0,C 180,E1 -2888.674,E2 -2888.674} C_VEL
LIN {X 0,Y 559.208,Z 717.639,A -85,B 0,C 180,E1 -2891.6,E2 -2891.6} C_VEL
LIN {X 0,Y 559.202,Z 717.634,A -85,B 0,C 180,E1 -2894.595,E2 -2894.595} C_VEL
LIN {X 0,Y 559.166,Z 717.644,A -85,B 0,C 180,E1 -2897.557,E2 -2897.557} C_VEL
LIN {X 0,Y 559.175,Z 717.646,A -85,B 0,C 180,E1 -2899.837,E2 -2899.837} C_VEL
LIN {X 0,Y 559.144,Z 717.648,A -85,B 0,C 180,E1 -2902.153,E2 -2902.153} C_VEL
LIN {X 0,Y 559.181,Z 717.638,A -85,B 0,C 180,E1 -2905.187,E2 -2905.187} C_VEL
LIN {X 0,Y 559.194,Z 717.64,A -85,B 0,C 180,E1 -2907.711,E2 -2907.711} C_VEL
LIN {X 0,Y 559.165,Z 717.639,A -85,B 0,C 180,E1 -2911.019,E2 -2911.019} C_VEL
LIN {X 0,Y 559.17,Z 717.645,A -85,B 0,C 180,E1 -2913.949,E2 -2913.949} C_VEL
LIN {X 0,Y 559.171,Z 717.641,A -85,B 0,C 180,E1 -2916.448,E2 -2916.448} C_VEL
LIN {X 0,Y 559.18,Z 717.629,A -85,B 0,C 180,E1 -2918.934,E2 -2918.934} C_VEL
LIN {X 0,Y 559.193,Z 717.634,A -85,B 0,C 180,E1 -2921.767,E2 -2921.767} C_VEL
LIN {X 0,Y 559.14,Z 717.647,A -85,B 0,C 180,E1 -2924.739,E2 -2924.739} C_VEL
LIN {X 0,Y 559.163,Z 717.638,A -85,B 0,C 180,E1 -2927.257,E2 -2927.257} C_VEL
LIN {X 0,Y 559.187,Z 717.639,A -85,B 0,C 180,E1 -2930.135,E2 -2930.135} C_VEL
LIN {X 0,Y 559.148,Z 717.645,A -85,B 0,C 180,E1 -2932.892,E2 -2932.892} C_VEL
LIN {X 0,Y 559.159,Z 717.64,A -85,B 0,C 180,E1 -2935.556,E2 -2935.556} C_VEL
LIN {X 0,Y 559.172,Z 717.64,A -85,B 0,C 180,E1 -2938.138,E2 -2938.138} C_VEL
LIN {X 0,Y 559.145,Z 717.648,A -85,B 0,C 180,E1 -2940.646,E2 -2940.646} C_VEL
LIN {X 0,Y 559.172,Z 717.642,A -85,B 0,C 180,E1 -2943.172,E2 -2943.172} C_VEL
LIN {X 0,Y 559.158,Z 717.641,A -85,B 0,C 180,E1 -2945.495,E2 -2945.495} C_VEL
LIN {X 0,Y 559.205,Z 717.853,A -85,B 0,C 180,E1 -2948.037,E2 -2948.037} C_VEL
LIN {X 0,Y 559.769,Z 723.25,A -85,B 0,C 180,E1 -2949.033,E2 -2949.033} C_VEL
LIN {X 0,Y 559.558,Z 739.471,A -85,B 0,C 180,E1 -2951.889,E2 -2951.889} C_VEL
LIN {X 0,Y 559.306,Z 756.882,A -85,B 0,C 180,E1 -2954.905,E2 -2954.905} C_VEL
LIN {X 0,Y 559.164,Z 771.914,A -85,B 0,C 180,E1 -2957.478,E2 -2957.478} C_VEL
LIN {X 0,Y 559.107,Z 779.997,A -85,B 0,C 180,E1 -2958.815,E2 -2958.815} C_VEL
LIN {X 0,Y 559.498,Z 783.301,A -85,B 0,C 180,E1 -2958.9,E2 -2958.9} C_VEL
LIN {X 0,Y 559.69,Z 798.068,A -85,B 0,C 180,E1 -2959.093,E2 -2959.093} C_VEL
LIN {X 0,Y 559.629,Z 856.138,A -85,B 0,C 180,E1 -2959.851,E2 -2959.851} C_VEL
LIN {X 0,Y 559.574,Z 865.412,A -85,B 0,C 180,E1 -2960.056,E2 -2960.056} C_VEL
LIN {X 0,Y 559.489,Z 873.89,A -85,B 0,C 180,E1 -2960.328,E2 -2960.328} C_VEL
LIN {X 0,Y 559.416,Z 882.398,A -85,B 0,C 180,E1 -2960.692,E2 -2960.692} C_VEL
LIN {X 0,Y 559.303,Z 890.731,A -85,B 0,C 180,E1 -2961.145,E2 -2961.145} C_VEL
LIN {X 0,Y 559.183,Z 898.769,A -85,B 0,C 180,E1 -2961.69,E2 -2961.69} C_VEL
LIN {X 0,Y 559.097,Z 907.431,A -85,B 0,C 180,E1 -2962.416,E2 -2962.416} C_VEL
LIN {X 0,Y 559.021,Z 915.824,A -85,B 0,C 180,E1 -2963.307,E2 -2963.307} C_VEL
LIN {X 0,Y 559.004,Z 921.434,A -85,B 0,C 180,E1 -2964.046,E2 -2964.046} C_VEL
LIN {X 0,Y 558.822,Z 926.988,A -85,B 0,C 180,E1 -2964.949,E2 -2964.949} C_VEL
LIN {X 0,Y 558.858,Z 932.148,A -85,B 0,C 180,E1 -2966.034,E2 -2966.034} C_VEL
LIN {X 0,Y 558.803,Z 935.935,A -85,B 0,C 180,E1 -2967.116,E2 -2967.116} C_VEL
LIN {X 0,Y 558.744,Z 937.682,A -85,B 0,C 180,E1 -2967.837,E2 -2967.837} C_VEL
LIN {X 0,Y 558.744,Z 938.935,A -85,B 0,C 180,E1 -2968.558,E2 -2968.558} C_VEL
LIN {X 0,Y 558.739,Z 939.71,A -85,B 0,C 180,E1 -2969.279,E2 -2969.279} C_VEL
LIN {X 0,Y 558.737,Z 940,A -85,B 0,C 180,E1 -2970,E2 -2970} C_VEL
LIN {X 0,Y 558.739,Z 939.71,A -85,B 0,C 180,E1 -2970.721,E2 -2970.721} C_VEL
LIN {X 0,Y 558.744,Z 938.935,A -85,B 0,C 180,E1 -2971.442,E2 -2971.442} C_VEL
LIN {X 0,Y 558.744,Z 937.681,A -85,B 0,C 180,E1 -2972.163,E2 -2972.163} C_VEL
LIN {X 0,Y 558.836,Z 934.788,A -85,B 0,C 180,E1 -2973.244,E2 -2973.244} C_VEL
LIN {X 0,Y 558.858,Z 932.148,A -85,B 0,C 180,E1 -2973.966,E2 -2973.966} C_VEL
LIN {X 0,Y 558.822,Z 926.985,A -85,B 0,C 180,E1 -2975.051,E2 -2975.051} C_VEL
LIN {X 0,Y 559.018,Z 920.186,A -85,B 0,C 180,E1 -2976.134,E2 -2976.134} C_VEL
LIN {X 0,Y 559.036,Z 912.744,A -85,B 0,C 180,E1 -2977.04,E2 -2977.04} C_VEL
LIN {X 0,Y 559.122,Z 905.406,A -85,B 0,C 180,E1 -2977.766,E2 -2977.766} C_VEL
LIN {X 0,Y 559.222,Z 897.544,A -85,B 0,C 180,E1 -2978.401,E2 -2978.401} C_VEL
LIN {X 0,Y 559.343,Z 887.73,A -85,B 0,C 180,E1 -2979.036,E2 -2979.036} C_VEL
LIN {X 0,Y 559.439,Z 876.302,A -85,B 0,C 180,E1 -2979.582,E2 -2979.582} C_VEL
LIN {X 0,Y 559.538,Z 866.245,A -85,B 0,C 180,E1 -2979.922,E2 -2979.922} C_VEL
LIN {X 0,Y 559.592,Z 857.441,A -85,B 0,C 180,E1 -2980.127,E2 -2980.127} C_VEL
LIN {X 0,Y 559.691,Z 798.099,A -85,B 0,C 180,E1 -2980.906,E2 -2980.906} C_VEL
LIN {X 0,Y 559.521,Z 783.575,A -85,B 0,C 180,E1 -2981.096,E2 -2981.096} C_VEL
LIN {X 0,Y 559.102,Z 780.03,A -85,B 0,C 180,E1 -2981.183,E2 -2981.183} C_VEL
LIN {X 0,Y 559.262,Z 764.344,A -85,B 0,C 180,E1 -2983.814,E2 -2983.814} C_VEL
LIN {X 0,Y 559.45,Z 747.041,A -85,B 0,C 180,E1 -2986.794,E2 -2986.794} C_VEL
LIN {X 0,Y 559.695,Z 729.738,A -85,B 0,C 180,E1 -2989.818,E2 -2989.818} C_VEL
LIN {X 0,Y 559.74,Z 721.087,A -85,B 0,C 180,E1 -2991.353,E2 -2991.353} C_VEL
LIN {X 0,Y 559.192,Z 717.673,A -85,B 0,C 180,E1 -2992.038,E2 -2992.038} C_VEL
LIN {X 0,Y 559.178,Z 717.646,A -85,B 0,C 180,E1 -2995.298,E2 -2995.298} C_VEL
LIN {X 0,Y 559.182,Z 717.641,A -85,B 0,C 180,E1 -2997.712,E2 -2997.712} C_VEL
LIN {X 0,Y 559.158,Z 717.637,A -85,B 0,C 180,E1 -3000.183,E2 -3000.183} C_VEL
LIN {X 0,Y 559.177,Z 717.639,A -85,B 0,C 180,E1 -3002.714,E2 -3002.714} C_VEL
LIN {X 0,Y 559.161,Z 717.649,A -85,B 0,C 180,E1 -3005.322,E2 -3005.322} C_VEL
LIN {X 0,Y 559.136,Z 717.645,A -85,B 0,C 180,E1 -3008.017,E2 -3008.017} C_VEL
LIN {X 0,Y 559.178,Z 717.636,A -85,B 0,C 180,E1 -3010.811,E2 -3010.811} C_VEL
LIN {X 0,Y 559.16,Z 717.648,A -85,B 0,C 180,E1 -3013.732,E2 -3013.732} C_VEL
LIN {X 0,Y 559.148,Z 717.641,A -85,B 0,C 180,E1 -3016.803,E2 -3016.803} C_VEL
LIN {X 0,Y 559.178,Z 717.636,A -85,B 0,C 180,E1 -3019.19,E2 -3019.19} C_VEL
LIN {X 0,Y 559.137,Z 717.645,A -85,B 0,C 180,E1 -3021.983,E2 -3021.983} C_VEL
LIN {X 0,Y 559.162,Z 717.639,A -85,B 0,C 180,E1 -3024.783,E2 -3024.783} C_VEL
LIN {X 0,Y 559.176,Z 717.641,A -85,B 0,C 180,E1 -3027.362,E2 -3027.362} C_VEL
LIN {X 0,Y 559.152,Z 717.645,A -85,B 0,C 180,E1 -3030.142,E2 -3030.142} C_VEL
LIN {X 0,Y 559.171,Z 717.638,A -85,B 0,C 180,E1 -3033.098,E2 -3033.098} C_VEL
LIN {X 0,Y 559.159,Z 717.642,A -85,B 0,C 180,E1 -3035.495,E2 -3035.495} C_VEL
LIN {X 0,Y 559.174,Z 717.637,A -85,B 0,C 180,E1 -3038.624,E2 -3038.624} C_VEL
LIN {X 0,Y 559.174,Z 717.638,A -85,B 0,C 180,E1 -3040.926,E2 -3040.926} C_VEL
LIN {X 0,Y 559.17,Z 717.645,A -85,B 0,C 180,E1 -3043.948,E2 -3043.948} C_VEL
LIN {X 0,Y 559.175,Z 717.646,A -85,B 0,C 180,E1 -3046.184,E2 -3046.184} C_VEL
LIN {X 0,Y 559.197,Z 717.633,A -85,B 0,C 180,E1 -3049.134,E2 -3049.134} C_VEL
LIN {X 0,Y 559.208,Z 717.639,A -85,B 0,C 180,E1 -3052.054,E2 -3052.054} C_VEL
LIN {X 0,Y 559.256,Z 717.628,A -85,B 0,C 180,E1 -3054.953,E2 -3054.953} C_VEL
LIN {X 0,Y 559.255,Z 717.624,A -85,B 0,C 180,E1 -3057.84,E2 -3057.84} C_VEL
LIN {X 0,Y 559.275,Z 717.632,A -85,B 0,C 180,E1 -3060.72,E2 -3060.72} C_VEL
LIN {X 0,Y 559.243,Z 717.634,A -85,B 0,C 180,E1 -3062.881,E2 -3062.881} C_VEL
LIN {X 0,Y 559.234,Z 717.629,A -85,B 0,C 180,E1 -3065.77,E2 -3065.77} C_VEL
LIN {X 0,Y 559.189,Z 717.642,A -85,B 0,C 180,E1 -3068.674,E2 -3068.674} C_VEL
LIN {X 0,Y 559.208,Z 717.634,A -85,B 0,C 180,E1 -3071.6,E2 -3071.6} C_VEL
LIN {X 0,Y 559.203,Z 717.641,A -85,B 0,C 180,E1 -3074.596,E2 -3074.596} C_VEL
LIN {X 0,Y 559.145,Z 717.639,A -85,B 0,C 180,E1 -3077.557,E2 -3077.557} C_VEL
LIN {X 0,Y 559.169,Z 717.638,A -85,B 0,C 180,E1 -3079.838,E2 -3079.838} C_VEL
LIN {X 0,Y 559.143,Z 717.642,A -85,B 0,C 180,E1 -3082.153,E2 -3082.153} C_VEL
LIN {X 0,Y 559.177,Z 717.64,A -85,B 0,C 180,E1 -3085.298,E2 -3085.298} C_VEL
LIN {X 0,Y 559.159,Z 717.641,A -85,B 0,C 180,E1 -3087.713,E2 -3087.713} C_VEL
LIN {X 0,Y 559.138,Z 717.645,A -85,B 0,C 180,E1 -3090.614,E2 -3090.614} C_VEL
LIN {X 0,Y 558.477,Z 717.733,A -85,B 0,C 180,E1 -3091.216,E2 -3091.216} C_VEL
LIN {X 0,Y 555.614,Z 718.09,A -85,B 0,C 180,E1 -3092.192,E2 -3092.192} C_VEL
LIN {X 0,Y 553.197,Z 718.388,A -85,B 0,C 180,E1 -3092.977,E2 -3092.977} C_VEL
LIN {X 0,Y 552.17,Z 718.513,A -85,B 0,C 180,E1 -3093.584,E2 -3093.584} C_VEL
LIN {X 0,Y 552.092,Z 718.52,A -85,B 0,C 180,E1 -3093.79,E2 -3093.79} C_VEL
LIN {X 0,Y 552.107,Z 718.521,A -85,B 0,C 180,E1 -3096.747,E2 -3096.747} C_VEL
LIN {X 0,Y 552.129,Z 718.519,A -85,B 0,C 180,E1 -3099.527,E2 -3099.527} C_VEL
LIN {X 0,Y 552.131,Z 718.505,A -85,B 0,C 180,E1 -3102.426,E2 -3102.426} C_VEL
LIN {X 0,Y 552.093,Z 718.529,A -85,B 0,C 180,E1 -3105.562,E2 -3105.562} C_VEL
LIN {X 0,Y 552.121,Z 718.517,A -85,B 0,C 180,E1 -3108.554,E2 -3108.554} C_VEL
LIN {X 0,Y 552.118,Z 718.522,A -85,B 0,C 180,E1 -3111.411,E2 -3111.411} C_VEL
LIN {X 0,Y 552.087,Z 718.524,A -85,B 0,C 180,E1 -3114.156,E2 -3114.156} C_VEL
LIN {X 0,Y 552.107,Z 718.519,A -85,B 0,C 180,E1 -3116.814,E2 -3116.814} C_VEL
LIN {X 0,Y 552.1,Z 718.522,A -85,B 0,C 180,E1 -3119.391,E2 -3119.391} C_VEL
LIN {X 0,Y 552.079,Z 718.531,A -85,B 0,C 180,E1 -3121.9,E2 -3121.9} C_VEL
LIN {X 0,Y 552.107,Z 718.52,A -85,B 0,C 180,E1 -3124.661,E2 -3124.661} C_VEL
LIN {X 0,Y 552.092,Z 718.525,A -85,B 0,C 180,E1 -3127.549,E2 -3127.549} C_VEL
LIN {X 0,Y 552.146,Z 718.522,A -85,B 0,C 180,E1 -3130.375,E2 -3130.375} C_VEL
LIN {X 0,Y 552.177,Z 718.627,A -85,B 0,C 180,E1 -3131.638,E2 -3131.638} C_VEL
LIN {X 0,Y 552.199,Z 726.346,A -85,B 0,C 180,E1 -3133.36,E2 -3133.36} C_VEL
LIN {X 0,Y 552.053,Z 738.532,A -85,B 0,C 180,E1 -3136.002,E2 -3136.002} C_VEL
LIN {X 0,Y 551.973,Z 751.432,A -85,B 0,C 180,E1 -3138.768,E2 -3138.768} C_VEL
LIN {X 0,Y 552.76,Z 758.547,A -85,B 0,C 180,E1 -3138.876,E2 -3138.876} C_VEL
LIN {X 0,Y 552.6,Z 826.22,A -85,B 0,C 180,E1 -3139.767,E2 -3139.767} C_VEL
LIN {X 0,Y 552.554,Z 835.471,A -85,B 0,C 180,E1 -3139.974,E2 -3139.974} C_VEL
LIN {X 0,Y 552.479,Z 845.143,A -85,B 0,C 180,E1 -3140.296,E2 -3140.296} C_VEL
LIN {X 0,Y 552.369,Z 855.217,A -85,B 0,C 180,E1 -3140.756,E2 -3140.756} C_VEL
LIN {X 0,Y 552.252,Z 865.709,A -85,B 0,C 180,E1 -3141.4,E2 -3141.4} C_VEL
LIN {X 0,Y 552.079,Z 873.884,A -85,B 0,C 180,E1 -3142.042,E2 -3142.042} C_VEL
LIN {X 0,Y 551.998,Z 880.626,A -85,B 0,C 180,E1 -3142.685,E2 -3142.685} C_VEL
LIN {X 0,Y 551.93,Z 887.01,A -85,B 0,C 180,E1 -3143.419,E2 -3143.419} C_VEL
LIN {X 0,Y 551.917,Z 892.321,A -85,B 0,C 180,E1 -3144.153,E2 -3144.153} C_VEL
LIN {X 0,Y 551.752,Z 896.752,A -85,B 0,C 180,E1 -3144.885,E2 -3144.885} C_VEL
LIN {X 0,Y 551.806,Z 900.445,A -85,B 0,C 180,E1 -3145.617,E2 -3145.617} C_VEL
LIN {X 0,Y 551.762,Z 904.647,A -85,B 0,C 180,E1 -3146.714,E2 -3146.714} C_VEL
LIN {X 0,Y 551.657,Z 907.586,A -85,B 0,C 180,E1 -3147.81,E2 -3147.81} C_VEL
LIN {X 0,Y 551.643,Z 908.875,A -85,B 0,C 180,E1 -3148.54,E2 -3148.54} C_VEL
LIN {X 0,Y 551.637,Z 909.69,A -85,B 0,C 180,E1 -3149.27,E2 -3149.27} C_VEL
LIN {X 0,Y 551.638,Z 909.996,A -85,B 0,C 180,E1 -3150,E2 -3150} C_VEL
LIN {X 0,Y 551.638,Z 909.73,A -85,B 0,C 180,E1 -3150.73,E2 -3150.73} C_VEL
LIN {X 0,Y 551.644,Z 908.994,A -85,B 0,C 180,E1 -3151.46,E2 -3151.46} C_VEL
LIN {X 0,Y 551.658,Z 907.783,A -85,B 0,C 180,E1 -3152.19,E2 -3152.19} C_VEL
LIN {X 0,Y 551.761,Z 904.932,A -85,B 0,C 180,E1 -3153.286,E2 -3153.286} C_VEL
LIN {X 0,Y 551.807,Z 900.819,A -85,B 0,C 180,E1 -3154.383,E2 -3154.383} C_VEL
LIN {X 0,Y 551.819,Z 895.239,A -85,B 0,C 180,E1 -3155.481,E2 -3155.481} C_VEL
LIN {X 0,Y 551.921,Z 888.863,A -85,B 0,C 180,E1 -3156.431,E2 -3156.431} C_VEL
LIN {X 0,Y 551.966,Z 883.164,A -85,B 0,C 180,E1 -3157.131,E2 -3157.131} C_VEL
LIN {X 0,Y 552.064,Z 875.906,A -85,B 0,C 180,E1 -3157.866,E2 -3157.866} C_VEL
LIN {X 0,Y 552.196,Z 868.145,A -85,B 0,C 180,E1 -3158.508,E2 -3158.508} C_VEL
LIN {X 0,Y 552.276,Z 859.961,A -85,B 0,C 180,E1 -3159.061,E2 -3159.061} C_VEL
LIN {X 0,Y 552.437,Z 849.562,A -85,B 0,C 180,E1 -3159.612,E2 -3159.612} C_VEL
LIN {X 0,Y 552.568,Z 837.877,A -85,B 0,C 180,E1 -3160.049,E2 -3160.049} C_VEL
LIN {X 0,Y 552.652,Z 827.377,A -85,B 0,C 180,E1 -3160.302,E2 -3160.302} C_VEL
LIN {X 0,Y 552.6,Z 756.079,A -85,B 0,C 180,E1 -3161.249,E2 -3161.249} C_VEL
LIN {X 0,Y 552.007,Z 751.818,A -85,B 0,C 180,E1 -3161.339,E2 -3161.339} C_VEL
LIN {X 0,Y 551.935,Z 750.675,A -85,B 0,C 180,E1 -3161.482,E2 -3161.482} C_VEL
LIN {X 0,Y 552.128,Z 735.466,A -85,B 0,C 180,E1 -3164.749,E2 -3164.749} C_VEL
LIN {X 0,Y 552.267,Z 721.533,A -85,B 0,C 180,E1 -3167.783,E2 -3167.783} C_VEL
LIN {X 0,Y 552.198,Z 718.611,A -85,B 0,C 180,E1 -3168.457,E2 -3168.457} C_VEL
LIN {X 0,Y 552.111,Z 718.522,A -85,B 0,C 180,E1 -3171.683,E2 -3171.683} C_VEL
LIN {X 0,Y 552.089,Z 718.527,A -85,B 0,C 180,E1 -3174.039,E2 -3174.039} C_VEL
LIN {X 0,Y 552.092,Z 718.522,A -85,B 0,C 180,E1 -3176.99,E2 -3176.99} C_VEL
LIN {X 0,Y 552.114,Z 718.524,A -85,B 0,C 180,E1 -3180.05,E2 -3180.05} C_VEL
LIN {X 0,Y 552.111,Z 718.521,A -85,B 0,C 180,E1 -3182.845,E2 -3182.845} C_VEL
LIN {X 0,Y 552.077,Z 718.523,A -85,B 0,C 180,E1 -3185.439,E2 -3185.439} C_VEL
LIN {X 0,Y 552.097,Z 718.519,A -85,B 0,C 180,E1 -3187.885,E2 -3187.885} C_VEL
LIN {X 0,Y 552.109,Z 718.525,A -85,B 0,C 180,E1 -3190.481,E2 -3190.481} C_VEL
LIN {X 0,Y 552.108,Z 718.519,A -85,B 0,C 180,E1 -3193.424,E2 -3193.424} C_VEL
LIN {X 0,Y 552.108,Z 718.521,A -85,B 0,C 180,E1 -3196.576,E2 -3196.576} C_VEL
LIN {X 0,Y 552.109,Z 718.515,A -85,B 0,C 180,E1 -3199.519,E2 -3199.519} C_VEL
LIN {X 0,Y 552.092,Z 718.523,A -85,B 0,C 180,E1 -3202.336,E2 -3202.336} C_VEL
LIN {X 0,Y 552.084,Z 718.526,A -85,B 0,C 180,E1 -3205.051,E2 -3205.051} C_VEL
LIN {X 0,Y 552.116,Z 718.516,A -85,B 0,C 180,E1 -3207.681,E2 -3207.681} C_VEL
LIN {X 0,Y 552.109,Z 718.519,A -85,B 0,C 180,E1 -3210.235,E2 -3210.235} C_VEL
LIN {X 0,Y 552.139,Z 718.521,A -85,B 0,C 180,E1 -3213,E2 -3213} C_VEL
LIN {X 0,Y 552.115,Z 718.524,A -85,B 0,C 180,E1 -3215.161,E2 -3215.161} C_VEL
LIN {X 0,Y 552.128,Z 718.517,A -85,B 0,C 180,E1 -3218.337,E2 -3218.337} C_VEL
LIN {X 0,Y 552.153,Z 718.515,A -85,B 0,C 180,E1 -3220.674,E2 -3220.674} C_VEL
LIN {X 0,Y 552.118,Z 718.517,A -85,B 0,C 180,E1 -3223.737,E2 -3223.737} C_VEL
LIN {X 0,Y 552.137,Z 718.515,A -85,B 0,C 180,E1 -3226.004,E2 -3226.004} C_VEL
LIN {X 0,Y 552.166,Z 718.516,A -85,B 0,C 180,E1 -3228.993,E2 -3228.993} C_VEL
LIN {X 0,Y 552.158,Z 718.508,A -85,B 0,C 180,E1 -3231.951,E2 -3231.951} C_VEL
LIN {X 0,Y 552.233,Z 718.503,A -85,B 0,C 180,E1 -3234.889,E2 -3234.889} C_VEL
LIN {X 0,Y 552.229,Z 718.508,A -85,B 0,C 180,E1 -3237.812,E2 -3237.812} C_VEL
LIN {X 0,Y 552.245,Z 718.499,A -85,B 0,C 180,E1 -3240.729,E2 -3240.729} C_VEL
LIN {X 0,Y 552.209,Z 718.501,A -85,B 0,C 180,E1 -3242.918,E2 -3242.918} C_VEL
LIN {X 0,Y 552.197,Z 718.514,A -85,B 0,C 180,E1 -3245.844,E2 -3245.844} C_VEL
LIN {X 0,Y 552.164,Z 718.511,A -85,B 0,C 180,E1 -3248.786,E2 -3248.786} C_VEL
LIN {X 0,Y 552.165,Z 718.516,A -85,B 0,C 180,E1 -3251.75,E2 -3251.75} C_VEL
LIN {X 0,Y 552.139,Z 718.513,A -85,B 0,C 180,E1 -3254.748,E2 -3254.748} C_VEL
LIN {X 0,Y 552.117,Z 718.526,A -85,B 0,C 180,E1 -3257.788,E2 -3257.788} C_VEL
LIN {X 0,Y 552.134,Z 718.518,A -85,B 0,C 180,E1 -3260.101,E2 -3260.101} C_VEL
LIN {X 0,Y 552.098,Z 718.521,A -85,B 0,C 180,E1 -3262.451,E2 -3262.451} C_VEL
LIN {X 0,Y 552.157,Z 718.513,A -85,B 0,C 180,E1 -3265.35,E2 -3265.35} C_VEL
LIN {X 0,Y 552.128,Z 718.523,A -85,B 0,C 180,E1 -3268.097,E2 -3268.097} C_VEL
LIN {X 0,Y 552.109,Z 718.52,A -85,B 0,C 180,E1 -3270.609,E2 -3270.609} C_VEL
LIN {X 0,Y 552.125,Z 718.516,A -85,B 0,C 180,E1 -3273.185,E2 -3273.185} C_VEL
LIN {X 0,Y 552.115,Z 718.52,A -85,B 0,C 180,E1 -3275.841,E2 -3275.841} C_VEL
LIN {X 0,Y 552.127,Z 718.505,A -85,B 0,C 180,E1 -3279.062,E2 -3279.062} C_VEL
LIN {X 0,Y 552.141,Z 718.51,A -85,B 0,C 180,E1 -3281.444,E2 -3281.444} C_VEL
LIN {X 0,Y 552.097,Z 718.528,A -85,B 0,C 180,E1 -3284.532,E2 -3284.532} C_VEL
LIN {X 0,Y 552.132,Z 718.513,A -85,B 0,C 180,E1 -3287.584,E2 -3287.584} C_VEL
LIN {X 0,Y 552.151,Z 718.521,A -85,B 0,C 180,E1 -3290.475,E2 -3290.475} C_VEL
LIN {X 0,Y 552.116,Z 718.517,A -85,B 0,C 180,E1 -3293.316,E2 -3293.316} C_VEL
LIN {X 0,Y 552.133,Z 718.517,A -85,B 0,C 180,E1 -3295.939,E2 -3295.939} C_VEL
LIN {X 0,Y 552.12,Z 718.523,A -85,B 0,C 180,E1 -3298.541,E2 -3298.541} C_VEL
LIN {X 0,Y 552.126,Z 718.518,A -85,B 0,C 180,E1 -3301.438,E2 -3301.438} C_VEL
LIN {X 0,Y 552.132,Z 718.519,A -85,B 0,C 180,E1 -3304.356,E2 -3304.356} C_VEL
LIN {X 0,Y 552.11,Z 718.527,A -85,B 0,C 180,E1 -3307.55,E2 -3307.55} C_VEL
LIN {X 0,Y 552.168,Z 718.686,A -85,B 0,C 180,E1 -3307.887,E2 -3307.887} C_VEL
LIN {X 0,Y 552.816,Z 723.25,A -85,B 0,C 180,E1 -3308.757,E2 -3308.757} C_VEL
LIN {X 0,Y 552.559,Z 738.39,A -85,B 0,C 180,E1 -3311.459,E2 -3311.459} C_VEL
LIN {X 0,Y 552.341,Z 754.611,A -85,B 0,C 180,E1 -3314.313,E2 -3314.313} C_VEL
LIN {X 0,Y 552.139,Z 769.751,A -85,B 0,C 180,E1 -3316.942,E2 -3316.942} C_VEL
LIN {X 0,Y 552.05,Z 779.964,A -85,B 0,C 180,E1 -3318.669,E2 -3318.669} C_VEL
LIN {X 0,Y 552.511,Z 783.828,A -85,B 0,C 180,E1 -3318.765,E2 -3318.765} C_VEL
LIN {X 0,Y 552.759,Z 795.79,A -85,B 0,C 180,E1 -3318.925,E2 -3318.925} C_VEL
LIN {X 0,Y 552.657,Z 856.138,A -85,B 0,C 180,E1 -3319.722,E2 -3319.722} C_VEL
LIN {X 0,Y 552.592,Z 865.412,A -85,B 0,C 180,E1 -3319.929,E2 -3319.929} C_VEL
LIN {X 0,Y 552.481,Z 873.889,A -85,B 0,C 180,E1 -3320.204,E2 -3320.204} C_VEL
LIN {X 0,Y 552.407,Z 882.396,A -85,B 0,C 180,E1 -3320.572,E2 -3320.572} C_VEL
LIN {X 0,Y 552.271,Z 890.729,A -85,B 0,C 180,E1 -3321.032,E2 -3321.032} C_VEL
LIN {X 0,Y 552.173,Z 898.769,A -85,B 0,C 180,E1 -3321.583,E2 -3321.583} C_VEL
LIN {X 0,Y 552.047,Z 907.431,A -85,B 0,C 180,E1 -3322.318,E2 -3322.318} C_VEL
LIN {X 0,Y 551.953,Z 916.432,A -85,B 0,C 180,E1 -3323.3,E2 -3323.3} C_VEL
LIN {X 0,Y 551.917,Z 922.611,A -85,B 0,C 180,E1 -3324.153,E2 -3324.153} C_VEL
LIN {X 0,Y 551.743,Z 926.988,A -85,B 0,C 180,E1 -3324.884,E2 -3324.884} C_VEL
LIN {X 0,Y 551.778,Z 932.148,A -85,B 0,C 180,E1 -3325.983,E2 -3325.983} C_VEL
LIN {X 0,Y 551.729,Z 935.935,A -85,B 0,C 180,E1 -3327.079,E2 -3327.079} C_VEL
LIN {X 0,Y 551.655,Z 937.682,A -85,B 0,C 180,E1 -3327.81,E2 -3327.81} C_VEL
LIN {X 0,Y 551.644,Z 938.934,A -85,B 0,C 180,E1 -3328.54,E2 -3328.54} C_VEL
LIN {X 0,Y 551.639,Z 939.709,A -85,B 0,C 180,E1 -3329.27,E2 -3329.27} C_VEL
LIN {X 0,Y 551.637,Z 940,A -85,B 0,C 180,E1 -3330,E2 -3330} C_VEL
LIN {X 0,Y 551.639,Z 939.709,A -85,B 0,C 180,E1 -3330.73,E2 -3330.73} C_VEL
LIN {X 0,Y 551.644,Z 938.934,A -85,B 0,C 180,E1 -3331.46,E2 -3331.46} C_VEL
LIN {X 0,Y 551.655,Z 937.681,A -85,B 0,C 180,E1 -3332.19,E2 -3332.19} C_VEL
LIN {X 0,Y 551.761,Z 934.787,A -85,B 0,C 180,E1 -3333.286,E2 -3333.286} C_VEL
LIN {X 0,Y 551.778,Z 932.148,A -85,B 0,C 180,E1 -3334.017,E2 -3334.017} C_VEL
LIN {X 0,Y 551.743,Z 926.986,A -85,B 0,C 180,E1 -3335.116,E2 -3335.116} C_VEL
LIN {X 0,Y 551.956,Z 920.4,A -85,B 0,C 180,E1 -3336.184,E2 -3336.184} C_VEL
LIN {X 0,Y 551.993,Z 912.744,A -85,B 0,C 180,E1 -3337.131,E2 -3337.131} C_VEL
LIN {X 0,Y 552.078,Z 905.405,A -85,B 0,C 180,E1 -3337.866,E2 -3337.866} C_VEL
LIN {X 0,Y 552.195,Z 897.542,A -85,B 0,C 180,E1 -3338.508,E2 -3338.508} C_VEL
LIN {X 0,Y 552.319,Z 887.729,A -85,B 0,C 180,E1 -3339.152,E2 -3339.152} C_VEL
LIN {X 0,Y 552.46,Z 876.303,A -85,B 0,C 180,E1 -3339.704,E2 -3339.704} C_VEL
LIN {X 0,Y 552.552,Z 866.245,A -85,B 0,C 180,E1 -3340.049,E2 -3340.049} C_VEL
LIN {X 0,Y 552.605,Z 857.44,A -85,B 0,C 180,E1 -3340.256,E2 -3340.256} C_VEL
LIN {X 0,Y 552.758,Z 803.762,A -85,B 0,C 180,E1 -3340.971,E2 -3340.971} C_VEL
LIN {X 0,Y 552.599,Z 784.579,A -85,B 0,C 180,E1 -3341.223,E2 -3341.223} C_VEL
LIN {X 0,Y 552.072,Z 780.263,A -85,B 0,C 180,E1 -3341.311,E2 -3341.311} C_VEL
LIN {X 0,Y 552.08,Z 777.321,A -85,B 0,C 180,E1 -3341.752,E2 -3341.752} C_VEL
LIN {X 0,Y 552.305,Z 758.937,A -85,B 0,C 180,E1 -3344.932,E2 -3344.932} C_VEL
LIN {X 0,Y 552.576,Z 740.553,A -85,B 0,C 180,E1 -3348.156,E2 -3348.156} C_VEL
LIN {X 0,Y 552.803,Z 724.331,A -85,B 0,C 180,E1 -3351.048,E2 -3351.048} C_VEL
LIN {X 0,Y 552.484,Z 720.355,A -85,B 0,C 180,E1 -3351.781,E2 -3351.781} C_VEL
LIN {X 0,Y 552.132,Z 718.582,A -85,B 0,C 180,E1 -3352.162,E2 -3352.162} C_VEL
LIN {X 0,Y 552.157,Z 718.52,A -85,B 0,C 180,E1 -3355.351,E2 -3355.351} C_VEL
LIN {X 0,Y 552.121,Z 718.518,A -85,B 0,C 180,E1 -3358.098,E2 -3358.098} C_VEL
LIN {X 0,Y 552.109,Z 718.516,A -85,B 0,C 180,E1 -3360.609,E2 -3360.609} C_VEL
LIN {X 0,Y 552.125,Z 718.523,A -85,B 0,C 180,E1 -3363.185,E2 -3363.185} C_VEL
LIN {X 0,Y 552.115,Z 718.52,A -85,B 0,C 180,E1 -3365.842,E2 -3365.842} C_VEL
LIN {X 0,Y 552.127,Z 718.52,A -85,B 0,C 180,E1 -3369.062,E2 -3369.062} C_VEL
LIN {X 0,Y 552.141,Z 718.519,A -85,B 0,C 180,E1 -3371.444,E2 -3371.444} C_VEL
LIN {X 0,Y 552.096,Z 718.52,A -85,B 0,C 180,E1 -3374.532,E2 -3374.532} C_VEL
LIN {X 0,Y 552.132,Z 718.523,A -85,B 0,C 180,E1 -3377.585,E2 -3377.585} C_VEL
LIN {X 0,Y 552.136,Z 718.503,A -85,B 0,C 180,E1 -3380.473,E2 -3380.473} C_VEL
LIN {X 0,Y 552.117,Z 718.516,A -85,B 0,C 180,E1 -3383.316,E2 -3383.316} C_VEL
LIN {X 0,Y 552.134,Z 718.524,A -85,B 0,C 180,E1 -3385.94,E2 -3385.94} C_VEL
LIN {X 0,Y 552.12,Z 718.517,A -85,B 0,C 180,E1 -3388.541,E2 -3388.541} C_VEL
LIN {X 0,Y 552.126,Z 718.516,A -85,B 0,C 180,E1 -3391.438,E2 -3391.438} C_VEL
LIN {X 0,Y 552.132,Z 718.52,A -85,B 0,C 180,E1 -3394.356,E2 -3394.356} C_VEL
LIN {X 0,Y 552.112,Z 718.517,A -85,B 0,C 180,E1 -3396.759,E2 -3396.759} C_VEL
LIN {X 0,Y 552.123,Z 718.513,A -85,B 0,C 180,E1 -3399.12,E2 -3399.12} C_VEL
LIN {X 0,Y 552.133,Z 718.515,A -85,B 0,C 180,E1 -3401.445,E2 -3401.445} C_VEL
LIN {X 0,Y 552.12,Z 718.52,A -85,B 0,C 180,E1 -3403.737,E2 -3403.737} C_VEL
LIN {X 0,Y 552.138,Z 718.52,A -85,B 0,C 180,E1 -3406.005,E2 -3406.005} C_VEL
LIN {X 0,Y 552.165,Z 718.51,A -85,B 0,C 180,E1 -3408.994,E2 -3408.994} C_VEL
LIN {X 0,Y 552.162,Z 718.515,A -85,B 0,C 180,E1 -3411.952,E2 -3411.952} C_VEL
LIN {X 0,Y 552.231,Z 718.504,A -85,B 0,C 180,E1 -3414.889,E2 -3414.889} C_VEL
LIN {X 0,Y 552.226,Z 718.499,A -85,B 0,C 180,E1 -3417.812,E2 -3417.812} C_VEL
LIN {X 0,Y 552.245,Z 718.508,A -85,B 0,C 180,E1 -3420.729,E2 -3420.729} C_VEL
LIN {X 0,Y 552.209,Z 718.51,A -85,B 0,C 180,E1 -3422.918,E2 -3422.918} C_VEL
LIN {X 0,Y 552.203,Z 718.505,A -85,B 0,C 180,E1 -3425.844,E2 -3425.844} C_VEL
LIN {X 0,Y 552.157,Z 718.519,A -85,B 0,C 180,E1 -3428.786,E2 -3428.786} C_VEL
LIN {X 0,Y 552.165,Z 718.511,A -85,B 0,C 180,E1 -3431.751,E2 -3431.751} C_VEL
LIN {X 0,Y 552.14,Z 718.524,A -85,B 0,C 180,E1 -3434.748,E2 -3434.748} C_VEL
LIN {X 0,Y 552.102,Z 718.515,A -85,B 0,C 180,E1 -3437.789,E2 -3437.789} C_VEL
LIN {X 0,Y 552.129,Z 718.515,A -85,B 0,C 180,E1 -3440.101,E2 -3440.101} C_VEL
LIN {X 0,Y 552.094,Z 718.523,A -85,B 0,C 180,E1 -3442.451,E2 -3442.451} C_VEL
LIN {X 0,Y 552.139,Z 718.516,A -85,B 0,C 180,E1 -3445.346,E2 -3445.346} C_VEL
LIN {X 0,Y 552.112,Z 718.517,A -85,B 0,C 180,E1 -3448.098,E2 -3448.098} C_VEL
LIN {X 0,Y 552.101,Z 718.522,A -85,B 0,C 180,E1 -3450.611,E2 -3450.611} C_VEL
LIN {X 0,Y 552.109,Z 718.525,A -85,B 0,C 180,E1 -3453.186,E2 -3453.186} C_VEL
LIN {X 0,Y 552.092,Z 718.52,A -85,B 0,C 180,E1 -3453.79,E2 -3453.79} C_VEL
LIN {X 0,Y 551.452,Z 718.6,A -85,B 0,C 180,E1 -3454.398,E2 -3454.398} C_VEL
LIN {X 0,Y 548.637,Z 718.959,A -85,B 0,C 180,E1 -3455.387,E2 -3455.387} C_VEL
LIN {X 0,Y 546.227,Z 719.256,A -85,B 0,C 180,E1 -3456.182,E2 -3456.182} C_VEL
LIN {X 0,Y 545.164,Z 719.387,A -85,B 0,C 180,E1 -3456.796,E2 -3456.796} C_VEL
LIN {X 0,Y 545.063,Z 719.402,A -85,B 0,C 180,E1 -3457.004,E2 -3457.004} C_VEL
LIN {X 0,Y 545.066,Z 719.392,A -85,B 0,C 180,E1 -3460.143,E2 -3460.143} C_VEL
LIN {X 0,Y 545.063,Z 719.385,A -85,B 0,C 180,E1 -3462.697,E2 -3462.697} C_VEL
LIN {X 0,Y 545.05,Z 719.401,A -85,B 0,C 180,E1 -3465.87,E2 -3465.87} C_VEL
LIN {X 0,Y 545.082,Z 719.395,A -85,B 0,C 180,E1 -3468.885,E2 -3468.885} C_VEL
LIN {X 0,Y 545.081,Z 719.391,A -85,B 0,C 180,E1 -3470.818,E2 -3470.818} C_VEL
LIN {X 0,Y 545.043,Z 719.406,A -85,B 0,C 180,E1 -3473.62,E2 -3473.62} C_VEL
LIN {X 0,Y 545.05,Z 719.399,A -85,B 0,C 180,E1 -3476.327,E2 -3476.327} C_VEL
LIN {X 0,Y 545.066,Z 719.394,A -85,B 0,C 180,E1 -3478.952,E2 -3478.952} C_VEL
LIN {X 0,Y 545.077,Z 719.401,A -85,B 0,C 180,E1 -3481.506,E2 -3481.506} C_VEL
LIN {X 0,Y 545.065,Z 719.404,A -85,B 0,C 180,E1 -3483.999,E2 -3483.999} C_VEL
LIN {X 0,Y 545.036,Z 719.401,A -85,B 0,C 180,E1 -3487.242,E2 -3487.242} C_VEL
LIN {X 0,Y 545.118,Z 719.397,A -85,B 0,C 180,E1 -3490.415,E2 -3490.415} C_VEL
LIN {X 0,Y 545.13,Z 719.51,A -85,B 0,C 180,E1 -3491.587,E2 -3491.587} C_VEL
LIN {X 0,Y 545.213,Z 726.349,A -85,B 0,C 180,E1 -3493.14,E2 -3493.14} C_VEL
LIN {X 0,Y 545.023,Z 738.534,A -85,B 0,C 180,E1 -3495.818,E2 -3495.818} C_VEL
LIN {X 0,Y 544.903,Z 751.393,A -85,B 0,C 180,E1 -3498.614,E2 -3498.614} C_VEL
LIN {X 0,Y 545.796,Z 758.768,A -85,B 0,C 180,E1 -3498.735,E2 -3498.735} C_VEL
LIN {X 0,Y 545.631,Z 826.253,A -85,B 0,C 180,E1 -3499.635,E2 -3499.635} C_VEL
LIN {X 0,Y 545.584,Z 835.492,A -85,B 0,C 180,E1 -3499.845,E2 -3499.845} C_VEL
LIN {X 0,Y 545.498,Z 845.158,A -85,B 0,C 180,E1 -3500.171,E2 -3500.171} C_VEL
LIN {X 0,Y 545.378,Z 855.232,A -85,B 0,C 180,E1 -3500.637,E2 -3500.637} C_VEL
LIN {X 0,Y 545.246,Z 865.714,A -85,B 0,C 180,E1 -3501.289,E2 -3501.289} C_VEL
LIN {X 0,Y 545.049,Z 873.889,A -85,B 0,C 180,E1 -3501.939,E2 -3501.939} C_VEL
LIN {X 0,Y 544.934,Z 880.63,A -85,B 0,C 180,E1 -3502.59,E2 -3502.59} C_VEL
LIN {X 0,Y 544.88,Z 887.014,A -85,B 0,C 180,E1 -3503.334,E2 -3503.334} C_VEL
LIN {X 0,Y 544.86,Z 892.325,A -85,B 0,C 180,E1 -3504.077,E2 -3504.077} C_VEL
LIN {X 0,Y 544.678,Z 896.756,A -85,B 0,C 180,E1 -3504.818,E2 -3504.818} C_VEL
LIN {X 0,Y 544.702,Z 901.966,A -85,B 0,C 180,E1 -3505.931,E2 -3505.931} C_VEL
LIN {X 0,Y 544.69,Z 904.649,A -85,B 0,C 180,E1 -3506.671,E2 -3506.671} C_VEL
LIN {X 0,Y 544.572,Z 907.587,A -85,B 0,C 180,E1 -3507.781,E2 -3507.781} C_VEL
LIN {X 0,Y 544.544,Z 908.875,A -85,B 0,C 180,E1 -3508.521,E2 -3508.521} C_VEL
LIN {X 0,Y 544.538,Z 909.69,A -85,B 0,C 180,E1 -3509.26,E2 -3509.26} C_VEL
LIN {X 0,Y 544.539,Z 909.996,A -85,B 0,C 180,E1 -3510,E2 -3510} C_VEL
LIN {X 0,Y 544.539,Z 909.729,A -85,B 0,C 180,E1 -3510.74,E2 -3510.74} C_VEL
LIN {X 0,Y 544.545,Z 908.992,A -85,B 0,C 180,E1 -3511.479,E2 -3511.479} C_VEL
LIN {X 0,Y 544.572,Z 907.783,A -85,B 0,C 180,E1 -3512.219,E2 -3512.219} C_VEL
LIN {X 0,Y 544.688,Z 904.929,A -85,B 0,C 180,E1 -3513.329,E2 -3513.329} C_VEL
LIN {X 0,Y 544.707,Z 900.816,A -85,B 0,C 180,E1 -3514.44,E2 -3514.44} C_VEL
LIN {X 0,Y 544.762,Z 895.236,A -85,B 0,C 180,E1 -3515.553,E2 -3515.553} C_VEL
LIN {X 0,Y 544.856,Z 889.446,A -85,B 0,C 180,E1 -3516.438,E2 -3516.438} C_VEL
LIN {X 0,Y 544.912,Z 883.157,A -85,B 0,C 180,E1 -3517.224,E2 -3517.224} C_VEL
LIN {X 0,Y 545.005,Z 875.897,A -85,B 0,C 180,E1 -3517.968,E2 -3517.968} C_VEL
LIN {X 0,Y 545.167,Z 868.134,A -85,B 0,C 180,E1 -3518.619,E2 -3518.619} C_VEL
LIN {X 0,Y 545.269,Z 859.949,A -85,B 0,C 180,E1 -3519.178,E2 -3519.178} C_VEL
LIN {X 0,Y 545.446,Z 849.548,A -85,B 0,C 180,E1 -3519.736,E2 -3519.736} C_VEL
LIN {X 0,Y 545.589,Z 837.858,A -85,B 0,C 180,E1 -3520.179,E2 -3520.179} C_VEL
LIN {X 0,Y 545.681,Z 828.644,A -85,B 0,C 180,E1 -3520.411,E2 -3520.411} C_VEL
LIN {X 0,Y 545.727,Z 804.022,A -85,B 0,C 180,E1 -3520.762,E2 -3520.762} C_VEL
LIN {X 0,Y 545.633,Z 756.71,A -85,B 0,C 180,E1 -3521.386,E2 -3521.386} C_VEL
LIN {X 0,Y 544.917,Z 751.706,A -85,B 0,C 180,E1 -3521.496,E2 -3521.496} C_VEL
LIN {X 0,Y 544.869,Z 750.689,A -85,B 0,C 180,E1 -3521.629,E2 -3521.629} C_VEL
LIN {X 0,Y 545.091,Z 735.463,A -85,B 0,C 180,E1 -3524.943,E2 -3524.943} C_VEL
LIN {X 0,Y 545.243,Z 721.53,A -85,B 0,C 180,E1 -3528.02,E2 -3528.02} C_VEL
LIN {X 0,Y 545.133,Z 719.492,A -85,B 0,C 180,E1 -3528.51,E2 -3528.51} C_VEL
LIN {X 0,Y 545.066,Z 719.397,A -85,B 0,C 180,E1 -3531.163,E2 -3531.163} C_VEL
LIN {X 0,Y 545.051,Z 719.4,A -85,B 0,C 180,E1 -3533.725,E2 -3533.725} C_VEL
LIN {X 0,Y 545.042,Z 719.406,A -85,B 0,C 180,E1 -3536.003,E2 -3536.003} C_VEL
LIN {X 0,Y 545.07,Z 719.399,A -85,B 0,C 180,E1 -3538.744,E2 -3538.744} C_VEL
LIN {X 0,Y 545.059,Z 719.395,A -85,B 0,C 180,E1 -3541.679,E2 -3541.679} C_VEL
LIN {X 0,Y 545.06,Z 719.406,A -85,B 0,C 180,E1 -3544.565,E2 -3544.565} C_VEL
LIN {X 0,Y 545.036,Z 719.397,A -85,B 0,C 180,E1 -3547.304,E2 -3547.304} C_VEL
LIN {X 0,Y 545.066,Z 719.396,A -85,B 0,C 180,E1 -3550.143,E2 -3550.143} C_VEL
LIN {X 0,Y 545.08,Z 719.396,A -85,B 0,C 180,E1 -3553.107,E2 -3553.107} C_VEL
LIN {X 0,Y 545.05,Z 719.397,A -85,B 0,C 180,E1 -3556.226,E2 -3556.226} C_VEL
LIN {X 0,Y 545.082,Z 719.397,A -85,B 0,C 180,E1 -3558.885,E2 -3558.885} C_VEL
LIN {X 0,Y 545.08,Z 719.402,A -85,B 0,C 180,E1 -3560.818,E2 -3560.818} C_VEL
LIN {X 0,Y 545.043,Z 719.399,A -85,B 0,C 180,E1 -3563.62,E2 -3563.62} C_VEL
LIN {X 0,Y 545.052,Z 719.398,A -85,B 0,C 180,E1 -3566.327,E2 -3566.327} C_VEL
LIN {X 0,Y 545.067,Z 719.405,A -85,B 0,C 180,E1 -3568.952,E2 -3568.952} C_VEL
LIN {X 0,Y 545.086,Z 719.395,A -85,B 0,C 180,E1 -3571.507,E2 -3571.507} C_VEL
LIN {X 0,Y 545.088,Z 719.391,A -85,B 0,C 180,E1 -3574.493,E2 -3574.493} C_VEL
LIN {X 0,Y 545.039,Z 719.407,A -85,B 0,C 180,E1 -3577.242,E2 -3577.242} C_VEL
LIN {X 0,Y 545.119,Z 719.389,A -85,B 0,C 180,E1 -3580.415,E2 -3580.415} C_VEL
LIN {X 0,Y 545.075,Z 719.396,A -85,B 0,C 180,E1 -3583.521,E2 -3583.521} C_VEL
LIN {X 0,Y 545.097,Z 719.393,A -85,B 0,C 180,E1 -3585.82,E2 -3585.82} C_VEL
LIN {X 0,Y 545.121,Z 719.392,A -85,B 0,C 180,E1 -3588.849,E2 -3588.849} C_VEL
LIN {X 0,Y 545.129,Z 719.384,A -85,B 0,C 180,E1 -3591.847,E2 -3591.847} C_VEL
LIN {X 0,Y 545.209,Z 719.377,A -85,B 0,C 180,E1 -3594.823,E2 -3594.823} C_VEL
LIN {X 0,Y 545.2,Z 719.384,A -85,B 0,C 180,E1 -3597.784,E2 -3597.784} C_VEL
LIN {X 0,Y 545.215,Z 719.375,A -85,B 0,C 180,E1 -3600.738,E2 -3600.738} C_VEL
LIN {X 0,Y 545.175,Z 719.377,A -85,B 0,C 180,E1 -3602.956,E2 -3602.956} C_VEL
LIN {X 0,Y 545.169,Z 719.388,A -85,B 0,C 180,E1 -3605.919,E2 -3605.919} C_VEL
LIN {X 0,Y 545.123,Z 719.389,A -85,B 0,C 180,E1 -3608.9,E2 -3608.9} C_VEL
LIN {X 0,Y 545.137,Z 719.39,A -85,B 0,C 180,E1 -3611.904,E2 -3611.904} C_VEL
LIN {X 0,Y 545.088,Z 719.392,A -85,B 0,C 180,E1 -3614.943,E2 -3614.943} C_VEL
LIN {X 0,Y 545.085,Z 719.4,A -85,B 0,C 180,E1 -3618.025,E2 -3618.025} C_VEL
LIN {X 0,Y 545.098,Z 719.39,A -85,B 0,C 180,E1 -3620.372,E2 -3620.372} C_VEL
LIN {X 0,Y 545.094,Z 719.394,A -85,B 0,C 180,E1 -3623.559,E2 -3623.559} C_VEL
LIN {X 0,Y 545.081,Z 719.404,A -85,B 0,C 180,E1 -3626,E2 -3626} C_VEL
LIN {X 0,Y 545.092,Z 719.39,A -85,B 0,C 180,E1 -3628.748,E2 -3628.748} C_VEL
LIN {X 0,Y 545.061,Z 719.398,A -85,B 0,C 180,E1 -3631.679,E2 -3631.679} C_VEL
LIN {X 0,Y 545.084,Z 719.397,A -85,B 0,C 180,E1 -3634.563,E2 -3634.563} C_VEL
LIN {X 0,Y 545.041,Z 719.393,A -85,B 0,C 180,E1 -3637.304,E2 -3637.304} C_VEL
LIN {X 0,Y 545.094,Z 719.386,A -85,B 0,C 180,E1 -3640.14,E2 -3640.14} C_VEL
LIN {X 0,Y 545.079,Z 719.394,A -85,B 0,C 180,E1 -3643.106,E2 -3643.106} C_VEL
LIN {X 0,Y 545.058,Z 719.403,A -85,B 0,C 180,E1 -3646.225,E2 -3646.225} C_VEL
LIN {X 0,Y 545.099,Z 719.393,A -85,B 0,C 180,E1 -3648.887,E2 -3648.887} C_VEL
LIN {X 0,Y 545.09,Z 719.399,A -85,B 0,C 180,E1 -3650.819,E2 -3650.819} C_VEL
LIN {X 0,Y 545.057,Z 719.395,A -85,B 0,C 180,E1 -3653.621,E2 -3653.621} C_VEL
LIN {X 0,Y 545.073,Z 719.4,A -85,B 0,C 180,E1 -3656.329,E2 -3656.329} C_VEL
LIN {X 0,Y 545.069,Z 719.396,A -85,B 0,C 180,E1 -3658.952,E2 -3658.952} C_VEL
LIN {X 0,Y 545.104,Z 719.393,A -85,B 0,C 180,E1 -3661.508,E2 -3661.508} C_VEL
LIN {X 0,Y 545.097,Z 719.397,A -85,B 0,C 180,E1 -3664.491,E2 -3664.491} C_VEL
LIN {X 0,Y 545.075,Z 719.422,A -85,B 0,C 180,E1 -3667.644,E2 -3667.644} C_VEL
LIN {X 0,Y 545.188,Z 719.941,A -85,B 0,C 180,E1 -3667.848,E2 -3667.848} C_VEL
LIN {X 0,Y 545.841,Z 725.413,A -85,B 0,C 180,E1 -3668.868,E2 -3668.868} C_VEL
LIN {X 0,Y 545.595,Z 741.634,A -85,B 0,C 180,E1 -3671.798,E2 -3671.798} C_VEL
LIN {X 0,Y 545.279,Z 760.018,A -85,B 0,C 180,E1 -3675.062,E2 -3675.062} C_VEL
LIN {X 0,Y 545.027,Z 777.321,A -85,B 0,C 180,E1 -3678.093,E2 -3678.093} C_VEL
LIN {X 0,Y 544.982,Z 780,A -85,B 0,C 180,E1 -3678.524,E2 -3678.524} C_VEL
LIN {X 0,Y 545.65,Z 785.207,A -85,B 0,C 180,E1 -3678.64,E2 -3678.64} C_VEL
LIN {X 0,Y 545.694,Z 856.138,A -85,B 0,C 180,E1 -3679.589,E2 -3679.589} C_VEL
LIN {X 0,Y 545.614,Z 865.411,A -85,B 0,C 180,E1 -3679.798,E2 -3679.798} C_VEL
LIN {X 0,Y 545.495,Z 873.887,A -85,B 0,C 180,E1 -3680.077,E2 -3680.077} C_VEL
LIN {X 0,Y 545.413,Z 882.394,A -85,B 0,C 180,E1 -3680.45,E2 -3680.45} C_VEL
LIN {X 0,Y 545.244,Z 890.727,A -85,B 0,C 180,E1 -3680.915,E2 -3680.915} C_VEL
LIN {X 0,Y 545.158,Z 898.767,A -85,B 0,C 180,E1 -3681.474,E2 -3681.474} C_VEL
LIN {X 0,Y 545.01,Z 907.431,A -85,B 0,C 180,E1 -3682.218,E2 -3682.218} C_VEL
LIN {X 0,Y 544.903,Z 916.081,A -85,B 0,C 180,E1 -3683.167,E2 -3683.167} C_VEL
LIN {X 0,Y 544.844,Z 922.611,A -85,B 0,C 180,E1 -3684.077,E2 -3684.077} C_VEL
LIN {X 0,Y 544.671,Z 926.988,A -85,B 0,C 180,E1 -3684.818,E2 -3684.818} C_VEL
LIN {X 0,Y 544.701,Z 932.149,A -85,B 0,C 180,E1 -3685.931,E2 -3685.931} C_VEL
LIN {X 0,Y 544.659,Z 935.936,A -85,B 0,C 180,E1 -3687.041,E2 -3687.041} C_VEL
LIN {X 0,Y 544.57,Z 937.682,A -85,B 0,C 180,E1 -3687.781,E2 -3687.781} C_VEL
LIN {X 0,Y 544.545,Z 938.933,A -85,B 0,C 180,E1 -3688.521,E2 -3688.521} C_VEL
LIN {X 0,Y 544.539,Z 939.709,A -85,B 0,C 180,E1 -3689.261,E2 -3689.261} C_VEL
LIN {X 0,Y 544.538,Z 940,A -85,B 0,C 180,E1 -3690,E2 -3690} C_VEL
LIN {X 0,Y 544.539,Z 939.708,A -85,B 0,C 180,E1 -3690.739,E2 -3690.739} C_VEL
LIN {X 0,Y 544.545,Z 938.933,A -85,B 0,C 180,E1 -3691.479,E2 -3691.479} C_VEL
LIN {X 0,Y 544.57,Z 937.682,A -85,B 0,C 180,E1 -3692.219,E2 -3692.219} C_VEL
LIN {X 0,Y 544.689,Z 934.787,A -85,B 0,C 180,E1 -3693.329,E2 -3693.329} C_VEL
LIN {X 0,Y 544.701,Z 932.148,A -85,B 0,C 180,E1 -3694.069,E2 -3694.069} C_VEL
LIN {X 0,Y 544.671,Z 926.986,A -85,B 0,C 180,E1 -3695.182,E2 -3695.182} C_VEL
LIN {X 0,Y 544.88,Z 920.957,A -85,B 0,C 180,E1 -3696.183,E2 -3696.183} C_VEL
LIN {X 0,Y 544.921,Z 912.744,A -85,B 0,C 180,E1 -3697.224,E2 -3697.224} C_VEL
LIN {X 0,Y 545.038,Z 905.403,A -85,B 0,C 180,E1 -3697.968,E2 -3697.968} C_VEL
LIN {X 0,Y 545.163,Z 897.54,A -85,B 0,C 180,E1 -3698.619,E2 -3698.619} C_VEL
LIN {X 0,Y 545.313,Z 887.727,A -85,B 0,C 180,E1 -3699.271,E2 -3699.271} C_VEL
LIN {X 0,Y 545.466,Z 876.304,A -85,B 0,C 180,E1 -3699.83,E2 -3699.83} C_VEL
LIN {X 0,Y 545.573,Z 866.245,A -85,B 0,C 180,E1 -3700.179,E2 -3700.179} C_VEL
LIN {X 0,Y 545.644,Z 857.439,A -85,B 0,C 180,E1 -3700.389,E2 -3700.389} C_VEL
LIN {X 0,Y 545.788,Z 796.39,A -85,B 0,C 180,E1 -3701.21,E2 -3701.21} C_VEL
LIN {X 0,Y 545.684,Z 785.545,A -85,B 0,C 180,E1 -3701.355,E2 -3701.355} C_VEL
LIN {X 0,Y 545.006,Z 780.119,A -85,B 0,C 180,E1 -3701.467,E2 -3701.467} C_VEL
LIN {X 0,Y 545.071,Z 772.996,A -85,B 0,C 180,E1 -3702.662,E2 -3702.662} C_VEL
LIN {X 0,Y 545.288,Z 757.856,A -85,B 0,C 180,E1 -3705.32,E2 -3705.32} C_VEL
LIN {X 0,Y 545.595,Z 741.634,A -85,B 0,C 180,E1 -3708.202,E2 -3708.202} C_VEL
LIN {X 0,Y 545.839,Z 725.413,A -85,B 0,C 180,E1 -3711.132,E2 -3711.132} C_VEL
LIN {X 0,Y 545.407,Z 721.033,A -85,B 0,C 180,E1 -3711.943,E2 -3711.943} C_VEL
LIN {X 0,Y 545.093,Z 719.514,A -85,B 0,C 180,E1 -3712.256,E2 -3712.256} C_VEL
LIN {X 0,Y 545.119,Z 719.399,A -85,B 0,C 180,E1 -3715.18,E2 -3715.18} C_VEL
LIN {X 0,Y 545.09,Z 719.398,A -85,B 0,C 180,E1 -3717.656,E2 -3717.656} C_VEL
LIN {X 0,Y 545.078,Z 719.39,A -85,B 0,C 180,E1 -3720.246,E2 -3720.246} C_VEL
LIN {X 0,Y 545.091,Z 719.397,A -85,B 0,C 180,E1 -3723.064,E2 -3723.064} C_VEL
LIN {X 0,Y 545.065,Z 719.4,A -85,B 0,C 180,E1 -3725.678,E2 -3725.678} C_VEL
LIN {X 0,Y 545.055,Z 719.398,A -85,B 0,C 180,E1 -3728.237,E2 -3728.237} C_VEL
LIN {X 0,Y 545.094,Z 719.389,A -85,B 0,C 180,E1 -3730.474,E2 -3730.474} C_VEL
LIN {X 0,Y 545.08,Z 719.395,A -85,B 0,C 180,E1 -3733.107,E2 -3733.107} C_VEL
LIN {X 0,Y 545.068,Z 719.396,A -85,B 0,C 180,E1 -3736.224,E2 -3736.224} C_VEL
LIN {X 0,Y 545.103,Z 719.386,A -85,B 0,C 180,E1 -3738.887,E2 -3738.887} C_VEL
LIN {X 0,Y 545.056,Z 719.396,A -85,B 0,C 180,E1 -3741.763,E2 -3741.763} C_VEL
LIN {X 0,Y 545.067,Z 719.395,A -85,B 0,C 180,E1 -3744.534,E2 -3744.534} C_VEL
LIN {X 0,Y 545.083,Z 719.395,A -85,B 0,C 180,E1 -3747.213,E2 -3747.213} C_VEL
LIN {X 0,Y 545.068,Z 719.403,A -85,B 0,C 180,E1 -3749.811,E2 -3749.811} C_VEL
LIN {X 0,Y 545.094,Z 719.396,A -85,B 0,C 180,E1 -3752.345,E2 -3752.345} C_VEL
LIN {X 0,Y 545.119,Z 719.389,A -85,B 0,C 180,E1 -3754.821,E2 -3754.821} C_VEL
LIN {X 0,Y 545.046,Z 719.396,A -85,B 0,C 180,E1 -3757.243,E2 -3757.243} C_VEL
LIN {X 0,Y 545.123,Z 719.393,A -85,B 0,C 180,E1 -3760.415,E2 -3760.415} C_VEL
LIN {X 0,Y 545.077,Z 719.396,A -85,B 0,C 180,E1 -3763.521,E2 -3763.521} C_VEL
LIN {X 0,Y 545.098,Z 719.394,A -85,B 0,C 180,E1 -3765.82,E2 -3765.82} C_VEL
LIN {X 0,Y 545.12,Z 719.388,A -85,B 0,C 180,E1 -3768.849,E2 -3768.849} C_VEL
LIN {X 0,Y 545.132,Z 719.39,A -85,B 0,C 180,E1 -3771.847,E2 -3771.847} C_VEL
LIN {X 0,Y 545.206,Z 719.38,A -85,B 0,C 180,E1 -3774.823,E2 -3774.823} C_VEL
LIN {X 0,Y 545.198,Z 719.374,A -85,B 0,C 180,E1 -3777.784,E2 -3777.784} C_VEL
LIN {X 0,Y 545.216,Z 719.383,A -85,B 0,C 180,E1 -3780.739,E2 -3780.739} C_VEL
LIN {X 0,Y 545.176,Z 719.386,A -85,B 0,C 180,E1 -3782.956,E2 -3782.956} C_VEL
LIN {X 0,Y 545.174,Z 719.381,A -85,B 0,C 180,E1 -3785.92,E2 -3785.92} C_VEL
LIN {X 0,Y 545.114,Z 719.394,A -85,B 0,C 180,E1 -3788.9,E2 -3788.9} C_VEL
LIN {X 0,Y 545.137,Z 719.387,A -85,B 0,C 180,E1 -3791.904,E2 -3791.904} C_VEL
LIN {X 0,Y 545.088,Z 719.398,A -85,B 0,C 180,E1 -3794.944,E2 -3794.944} C_VEL
LIN {X 0,Y 545.074,Z 719.391,A -85,B 0,C 180,E1 -3798.026,E2 -3798.026} C_VEL
LIN {X 0,Y 545.095,Z 719.393,A -85,B 0,C 180,E1 -3800.372,E2 -3800.372} C_VEL
LIN {X 0,Y 545.081,Z 719.394,A -85,B 0,C 180,E1 -3803.559,E2 -3803.559} C_VEL
LIN {X 0,Y 545.08,Z 719.389,A -85,B 0,C 180,E1 -3806.001,E2 -3806.001} C_VEL
LIN {X 0,Y 545.091,Z 719.396,A -85,B 0,C 180,E1 -3808.748,E2 -3808.748} C_VEL
LIN {X 0,Y 545.057,Z 719.396,A -85,B 0,C 180,E1 -3811.915,E2 -3811.915} C_VEL
LIN {X 0,Y 545.061,Z 719.395,A -85,B 0,C 180,E1 -3814.565,E2 -3814.565} C_VEL
LIN {X 0,Y 545.063,Z 719.402,A -85,B 0,C 180,E1 -3817.004,E2 -3817.004} C_VEL
LIN {X 0,Y 544.355,Z 719.494,A -85,B 0,C 180,E1 -3817.62,E2 -3817.62} C_VEL
LIN {X 0,Y 541.489,Z 719.848,A -85,B 0,C 180,E1 -3818.621,E2 -3818.621} C_VEL
LIN {X 0,Y 539.101,Z 720.143,A -85,B 0,C 180,E1 -3819.427,E2 -3819.427} C_VEL
LIN {X 0,Y 538.092,Z 720.261,A -85,B 0,C 180,E1 -3820.049,E2 -3820.049} C_VEL
LIN {X 0,Y 538.017,Z 720.269,A -85,B 0,C 180,E1 -3820.26,E2 -3820.26} C_VEL
LIN {X 0,Y 538.007,Z 720.265,A -85,B 0,C 180,E1 -3822.985,E2 -3822.985} C_VEL
LIN {X 0,Y 538.02,Z 720.276,A -85,B 0,C 180,E1 -3825.927,E2 -3825.927} C_VEL
LIN {X 0,Y 538.031,Z 720.273,A -85,B 0,C 180,E1 -3828.227,E2 -3828.227} C_VEL
LIN {X 0,Y 538.014,Z 720.274,A -85,B 0,C 180,E1 -3831.17,E2 -3831.17} C_VEL
LIN {X 0,Y 537.996,Z 720.281,A -85,B 0,C 180,E1 -3834.089,E2 -3834.089} C_VEL
LIN {X 0,Y 538.032,Z 720.272,A -85,B 0,C 180,E1 -3836.727,E2 -3836.727} C_VEL
LIN {X 0,Y 538.016,Z 720.278,A -85,B 0,C 180,E1 -3839.558,E2 -3839.558} C_VEL
LIN {X 0,Y 538.016,Z 720.282,A -85,B 0,C 180,E1 -3841.949,E2 -3841.949} C_VEL
LIN {X 0,Y 538.041,Z 720.273,A -85,B 0,C 180,E1 -3844.466,E2 -3844.466} C_VEL
LIN {X 0,Y 538.013,Z 720.274,A -85,B 0,C 180,E1 -3846.928,E2 -3846.928} C_VEL
LIN {X 0,Y 538.082,Z 720.274,A -85,B 0,C 180,E1 -3850.148,E2 -3850.148} C_VEL
LIN {X 0,Y 538.118,Z 720.393,A -85,B 0,C 180,E1 -3851.536,E2 -3851.536} C_VEL
LIN {X 0,Y 538.124,Z 728.092,A -85,B 0,C 180,E1 -3853.302,E2 -3853.302} C_VEL
LIN {X 0,Y 537.962,Z 740.278,A -85,B 0,C 180,E1 -3856.014,E2 -3856.014} C_VEL
LIN {X 0,Y 537.874,Z 751.477,A -85,B 0,C 180,E1 -3858.459,E2 -3858.459} C_VEL
LIN {X 0,Y 538.843,Z 760.065,A -85,B 0,C 180,E1 -3858.604,E2 -3858.604} C_VEL
LIN {X 0,Y 538.661,Z 826.286,A -85,B 0,C 180,E1 -3859.499,E2 -3859.499} C_VEL
LIN {X 0,Y 538.603,Z 835.513,A -85,B 0,C 180,E1 -3859.712,E2 -3859.712} C_VEL
LIN {X 0,Y 538.507,Z 845.172,A -85,B 0,C 180,E1 -3860.042,E2 -3860.042} C_VEL
LIN {X 0,Y 538.386,Z 855.246,A -85,B 0,C 180,E1 -3860.514,E2 -3860.514} C_VEL
LIN {X 0,Y 538.23,Z 865.72,A -85,B 0,C 180,E1 -3861.174,E2 -3861.174} C_VEL
LIN {X 0,Y 538.015,Z 873.894,A -85,B 0,C 180,E1 -3861.833,E2 -3861.833} C_VEL
LIN {X 0,Y 537.885,Z 880.635,A -85,B 0,C 180,E1 -3862.492,E2 -3862.492} C_VEL
LIN {X 0,Y 537.824,Z 887.273,A -85,B 0,C 180,E1 -3863.28,E2 -3863.28} C_VEL
LIN {X 0,Y 537.785,Z 892.328,A -85,B 0,C 180,E1 -3863.999,E2 -3863.999} C_VEL
LIN {X 0,Y 537.61,Z 896.759,A -85,B 0,C 180,E1 -3864.75,E2 -3864.75} C_VEL
LIN {X 0,Y 537.625,Z 901.968,A -85,B 0,C 180,E1 -3865.877,E2 -3865.877} C_VEL
LIN {X 0,Y 537.589,Z 904.65,A -85,B 0,C 180,E1 -3866.627,E2 -3866.627} C_VEL
LIN {X 0,Y 537.491,Z 907.588,A -85,B 0,C 180,E1 -3867.752,E2 -3867.752} C_VEL
LIN {X 0,Y 537.45,Z 908.875,A -85,B 0,C 180,E1 -3868.501,E2 -3868.501} C_VEL
LIN {X 0,Y 537.438,Z 909.69,A -85,B 0,C 180,E1 -3869.251,E2 -3869.251} C_VEL
LIN {X 0,Y 537.44,Z 909.996,A -85,B 0,C 180,E1 -3870,E2 -3870} C_VEL
LIN {X 0,Y 537.439,Z 909.728,A -85,B 0,C 180,E1 -3870.749,E2 -3870.749} C_VEL
LIN {X 0,Y 537.451,Z 908.991,A -85,B 0,C 180,E1 -3871.499,E2 -3871.499} C_VEL
LIN {X 0,Y 537.491,Z 907.782,A -85,B 0,C 180,E1 -3872.248,E2 -3872.248} C_VEL
LIN {X 0,Y 537.587,Z 904.927,A -85,B 0,C 180,E1 -3873.373,E2 -3873.373} C_VEL
LIN {X 0,Y 537.621,Z 902.332,A -85,B 0,C 180,E1 -3874.123,E2 -3874.123} C_VEL
LIN {X 0,Y 537.602,Z 897.217,A -85,B 0,C 180,E1 -3875.25,E2 -3875.25} C_VEL
LIN {X 0,Y 537.803,Z 891.504,A -85,B 0,C 180,E1 -3876.223,E2 -3876.223} C_VEL
LIN {X 0,Y 537.849,Z 883.152,A -85,B 0,C 180,E1 -3877.319,E2 -3877.319} C_VEL
LIN {X 0,Y 537.984,Z 875.889,A -85,B 0,C 180,E1 -3878.073,E2 -3878.073} C_VEL
LIN {X 0,Y 538.146,Z 868.124,A -85,B 0,C 180,E1 -3878.732,E2 -3878.732} C_VEL
LIN {X 0,Y 538.275,Z 859.937,A -85,B 0,C 180,E1 -3879.298,E2 -3879.298} C_VEL
LIN {X 0,Y 538.436,Z 849.534,A -85,B 0,C 180,E1 -3879.864,E2 -3879.864} C_VEL
LIN {X 0,Y 538.613,Z 837.839,A -85,B 0,C 180,E1 -3880.312,E2 -3880.312} C_VEL
LIN {X 0,Y 538.706,Z 828.612,A -85,B 0,C 180,E1 -3880.548,E2 -3880.548} C_VEL
LIN {X 0,Y 538.77,Z 802.188,A -85,B 0,C 180,E1 -3880.927,E2 -3880.927} C_VEL
LIN {X 0,Y 538.675,Z 757.102,A -85,B 0,C 180,E1 -3881.529,E2 -3881.529} C_VEL
LIN {X 0,Y 537.879,Z 752.033,A -85,B 0,C 180,E1 -3881.63,E2 -3881.63} C_VEL
LIN {X 0,Y 537.807,Z 750.808,A -85,B 0,C 180,E1 -3881.758,E2 -3881.758} C_VEL
LIN {X 0,Y 538.038,Z 736.792,A -85,B 0,C 180,E1 -3884.848,E2 -3884.848} C_VEL
LIN {X 0,Y 538.208,Z 723.443,A -85,B 0,C 180,E1 -3887.831,E2 -3887.831} C_VEL
LIN {X 0,Y 538.087,Z 720.376,A -85,B 0,C 180,E1 -3888.564,E2 -3888.564} C_VEL
LIN {X 0,Y 538.038,Z 720.275,A -85,B 0,C 180,E1 -3890.651,E2 -3890.651} C_VEL
LIN {X 0,Y 538.008,Z 720.279,A -85,B 0,C 180,E1 -3893.878,E2 -3893.878} C_VEL
LIN {X 0,Y 538.007,Z 720.284,A -85,B 0,C 180,E1 -3896.369,E2 -3896.369} C_VEL
LIN {X 0,Y 538.031,Z 720.274,A -85,B 0,C 180,E1 -3898.933,E2 -3898.933} C_VEL
LIN {X 0,Y 538.011,Z 720.275,A -85,B 0,C 180,E1 -3901.887,E2 -3901.887} C_VEL
LIN {X 0,Y 538.01,Z 720.283,A -85,B 0,C 180,E1 -3904.617,E2 -3904.617} C_VEL
LIN {X 0,Y 538.005,Z 720.273,A -85,B 0,C 180,E1 -3907.17,E2 -3907.17} C_VEL
LIN {X 0,Y 538.012,Z 720.271,A -85,B 0,C 180,E1 -3909.798,E2 -3909.798} C_VEL
LIN {X 0,Y 538.02,Z 720.28,A -85,B 0,C 180,E1 -3912.786,E2 -3912.786} C_VEL
LIN {X 0,Y 538.019,Z 720.27,A -85,B 0,C 180,E1 -3915.927,E2 -3915.927} C_VEL
LIN {X 0,Y 538.049,Z 720.267,A -85,B 0,C 180,E1 -3919.253,E2 -3919.253} C_VEL
LIN {X 0,Y 537.992,Z 720.278,A -85,B 0,C 180,E1 -3922.122,E2 -3922.122} C_VEL
LIN {X 0,Y 537.999,Z 720.283,A -85,B 0,C 180,E1 -3924.916,E2 -3924.916} C_VEL
LIN {X 0,Y 538.019,Z 720.273,A -85,B 0,C 180,E1 -3927.617,E2 -3927.617} C_VEL
LIN {X 0,Y 538.015,Z 720.275,A -85,B 0,C 180,E1 -3930.239,E2 -3930.239} C_VEL
LIN {X 0,Y 538.058,Z 720.275,A -85,B 0,C 180,E1 -3932.796,E2 -3932.796} C_VEL
LIN {X 0,Y 538.045,Z 720.275,A -85,B 0,C 180,E1 -3935.292,E2 -3935.292} C_VEL
LIN {X 0,Y 538.024,Z 720.275,A -85,B 0,C 180,E1 -3938.546,E2 -3938.546} C_VEL
LIN {X 0,Y 538.036,Z 720.277,A -85,B 0,C 180,E1 -3940.94,E2 -3940.94} C_VEL
LIN {X 0,Y 538.023,Z 720.278,A -85,B 0,C 180,E1 -3943.299,E2 -3943.299} C_VEL
LIN {X 0,Y 538.066,Z 720.271,A -85,B 0,C 180,E1 -3945.631,E2 -3945.631} C_VEL
LIN {X 0,Y 538.08,Z 720.268,A -85,B 0,C 180,E1 -3948.702,E2 -3948.702} C_VEL
LIN {X 0,Y 538.086,Z 720.262,A -85,B 0,C 180,E1 -3951.74,E2 -3951.74} C_VEL
LIN {X 0,Y 538.166,Z 720.254,A -85,B 0,C 180,E1 -3954.755,E2 -3954.755} C_VEL
LIN {X 0,Y 538.172,Z 720.26,A -85,B 0,C 180,E1 -3957.755,E2 -3957.755} C_VEL
LIN {X 0,Y 538.185,Z 720.25,A -85,B 0,C 180,E1 -3960.748,E2 -3960.748} C_VEL
LIN {X 0,Y 538.142,Z 720.253,A -85,B 0,C 180,E1 -3962.994,E2 -3962.994} C_VEL
LIN {X 0,Y 538.123,Z 720.265,A -85,B 0,C 180,E1 -3965.997,E2 -3965.997} C_VEL
LIN {X 0,Y 538.074,Z 720.267,A -85,B 0,C 180,E1 -3969.017,E2 -3969.017} C_VEL
LIN {X 0,Y 538.086,Z 720.265,A -85,B 0,C 180,E1 -3972.062,E2 -3972.062} C_VEL
LIN {X 0,Y 538.048,Z 720.27,A -85,B 0,C 180,E1 -3975.144,E2 -3975.144} C_VEL
LIN {X 0,Y 538.037,Z 720.274,A -85,B 0,C 180,E1 -3978.27,E2 -3978.27} C_VEL
LIN {X 0,Y 538.042,Z 720.267,A -85,B 0,C 180,E1 -3980.651,E2 -3980.651} C_VEL
LIN {X 0,Y 538.027,Z 720.279,A -85,B 0,C 180,E1 -3983.887,E2 -3983.887} C_VEL
LIN {X 0,Y 538.044,Z 720.275,A -85,B 0,C 180,E1 -3986.366,E2 -3986.366} C_VEL
LIN {X 0,Y 538.033,Z 720.268,A -85,B 0,C 180,E1 -3988.934,E2 -3988.934} C_VEL
LIN {X 0,Y 538.016,Z 720.278,A -85,B 0,C 180,E1 -3991.888,E2 -3991.888} C_VEL
LIN {X 0,Y 538.034,Z 720.274,A -85,B 0,C 180,E1 -3994.621,E2 -3994.621} C_VEL
LIN {X 0,Y 538.009,Z 720.269,A -85,B 0,C 180,E1 -3997.17,E2 -3997.17} C_VEL
LIN {X 0,Y 538.056,Z 720.257,A -85,B 0,C 180,E1 -3999.794,E2 -3999.794} C_VEL
LIN {X 0,Y 538.02,Z 720.276,A -85,B 0,C 180,E1 -4002.786,E2 -4002.786} C_VEL
LIN {X 0,Y 538.033,Z 720.273,A -85,B 0,C 180,E1 -4005.141,E2 -4005.141} C_VEL
LIN {X 0,Y 538.042,Z 720.274,A -85,B 0,C 180,E1 -4008.228,E2 -4008.228} C_VEL
LIN {X 0,Y 538.02,Z 720.275,A -85,B 0,C 180,E1 -4011.17,E2 -4011.17} C_VEL
LIN {X 0,Y 538.031,Z 720.273,A -85,B 0,C 180,E1 -4014.083,E2 -4014.083} C_VEL
LIN {X 0,Y 538.033,Z 720.28,A -85,B 0,C 180,E1 -4016.728,E2 -4016.728} C_VEL
LIN {X 0,Y 538.027,Z 720.269,A -85,B 0,C 180,E1 -4019.556,E2 -4019.556} C_VEL
LIN {X 0,Y 538.045,Z 720.272,A -85,B 0,C 180,E1 -4021.95,E2 -4021.95} C_VEL
LIN {X 0,Y 538.073,Z 720.272,A -85,B 0,C 180,E1 -4024.467,E2 -4024.467} C_VEL
LIN {X 0,Y 538.045,Z 720.415,A -85,B 0,C 180,E1 -4027.639,E2 -4027.639} C_VEL
LIN {X 0,Y 538.854,Z 726.367,A -85,B 0,C 180,E1 -4028.781,E2 -4028.781} C_VEL
LIN {X 0,Y 538.584,Z 742.716,A -85,B 0,C 180,E1 -4031.749,E2 -4031.749} C_VEL
LIN {X 0,Y 538.246,Z 760.018,A -85,B 0,C 180,E1 -4034.862,E2 -4034.862} C_VEL
LIN {X 0,Y 537.987,Z 777.321,A -85,B 0,C 180,E1 -4037.935,E2 -4037.935} C_VEL
LIN {X 0,Y 537.964,Z 779.972,A -85,B 0,C 180,E1 -4038.372,E2 -4038.372} C_VEL
LIN {X 0,Y 538.643,Z 785.338,A -85,B 0,C 180,E1 -4038.492,E2 -4038.492} C_VEL
LIN {X 0,Y 538.826,Z 800.467,A -85,B 0,C 180,E1 -4038.697,E2 -4038.697} C_VEL
LIN {X 0,Y 538.735,Z 856.138,A -85,B 0,C 180,E1 -4039.453,E2 -4039.453} C_VEL
LIN {X 0,Y 538.638,Z 865.41,A -85,B 0,C 180,E1 -4039.665,E2 -4039.665} C_VEL
LIN {X 0,Y 538.519,Z 873.886,A -85,B 0,C 180,E1 -4039.947,E2 -4039.947} C_VEL
LIN {X 0,Y 538.398,Z 882.392,A -85,B 0,C 180,E1 -4040.325,E2 -4040.325} C_VEL
LIN {X 0,Y 538.237,Z 890.725,A -85,B 0,C 180,E1 -4040.796,E2 -4040.796} C_VEL
LIN {X 0,Y 538.137,Z 898.765,A -85,B 0,C 180,E1 -4041.362,E2 -4041.362} C_VEL
LIN {X 0,Y 537.971,Z 907.432,A -85,B 0,C 180,E1 -4042.116,E2 -4042.116} C_VEL
LIN {X 0,Y 537.858,Z 915.938,A -85,B 0,C 180,E1 -4043.058,E2 -4043.058} C_VEL
LIN {X 0,Y 537.772,Z 922.611,A -85,B 0,C 180,E1 -4043.999,E2 -4043.999} C_VEL
LIN {X 0,Y 537.604,Z 926.989,A -85,B 0,C 180,E1 -4044.75,E2 -4044.75} C_VEL
LIN {X 0,Y 537.624,Z 932.149,A -85,B 0,C 180,E1 -4045.877,E2 -4045.877} C_VEL
LIN {X 0,Y 537.562,Z 935.936,A -85,B 0,C 180,E1 -4047.002,E2 -4047.002} C_VEL
LIN {X 0,Y 537.489,Z 937.682,A -85,B 0,C 180,E1 -4047.752,E2 -4047.752} C_VEL
LIN {X 0,Y 537.45,Z 938.932,A -85,B 0,C 180,E1 -4048.501,E2 -4048.501} C_VEL
LIN {X 0,Y 537.44,Z 939.708,A -85,B 0,C 180,E1 -4049.251,E2 -4049.251} C_VEL
LIN {X 0,Y 537.439,Z 940,A -85,B 0,C 180,E1 -4050,E2 -4050} C_VEL
LIN {X 0,Y 537.44,Z 939.708,A -85,B 0,C 180,E1 -4050.749,E2 -4050.749} C_VEL
LIN {X 0,Y 537.45,Z 938.931,A -85,B 0,C 180,E1 -4051.499,E2 -4051.499} C_VEL
LIN {X 0,Y 537.489,Z 937.682,A -85,B 0,C 180,E1 -4052.248,E2 -4052.248} C_VEL
LIN {X 0,Y 537.588,Z 934.787,A -85,B 0,C 180,E1 -4053.373,E2 -4053.373} C_VEL
LIN {X 0,Y 537.624,Z 932.148,A -85,B 0,C 180,E1 -4054.123,E2 -4054.123} C_VEL
LIN {X 0,Y 537.604,Z 926.986,A -85,B 0,C 180,E1 -4055.25,E2 -4055.25} C_VEL
LIN {X 0,Y 537.802,Z 921.199,A -85,B 0,C 180,E1 -4056.226,E2 -4056.226} C_VEL
LIN {X 0,Y 537.853,Z 914.435,A -85,B 0,C 180,E1 -4057.131,E2 -4057.131} C_VEL
LIN {X 0,Y 537.992,Z 906.422,A -85,B 0,C 180,E1 -4057.978,E2 -4057.978} C_VEL
LIN {X 0,Y 538.137,Z 898.769,A -85,B 0,C 180,E1 -4058.638,E2 -4058.638} C_VEL
LIN {X 0,Y 538.237,Z 890.726,A -85,B 0,C 180,E1 -4059.204,E2 -4059.204} C_VEL
LIN {X 0,Y 538.398,Z 882.394,A -85,B 0,C 180,E1 -4059.675,E2 -4059.675} C_VEL
LIN {X 0,Y 538.519,Z 873.888,A -85,B 0,C 180,E1 -4060.053,E2 -4060.053} C_VEL
LIN {X 0,Y 538.603,Z 863.75,A -85,B 0,C 180,E1 -4060.383,E2 -4060.383} C_VEL
LIN {X 0,Y 538.767,Z 852.057,A -85,B 0,C 180,E1 -4060.618,E2 -4060.618} C_VEL
LIN {X 0,Y 538.773,Z 786.44,A -85,B 0,C 180,E1 -4061.491,E2 -4061.491} C_VEL
LIN {X 0,Y 537.995,Z 780.261,A -85,B 0,C 180,E1 -4061.609,E2 -4061.609} C_VEL
LIN {X 0,Y 537.987,Z 777.321,A -85,B 0,C 180,E1 -4062.065,E2 -4062.065} C_VEL
LIN {X 0,Y 538.246,Z 760.018,A -85,B 0,C 180,E1 -4065.138,E2 -4065.138} C_VEL
LIN {X 0,Y 538.584,Z 742.715,A -85,B 0,C 180,E1 -4068.251,E2 -4068.251} C_VEL
LIN {X 0,Y 538.851,Z 726.367,A -85,B 0,C 180,E1 -4071.219,E2 -4071.219} C_VEL
LIN {X 0,Y 538.108,Z 720.625,A -85,B 0,C 180,E1 -4072.307,E2 -4072.307} C_VEL
LIN {X 0,Y 538.035,Z 720.295,A -85,B 0,C 180,E1 -4072.462,E2 -4072.462} C_VEL
LIN {X 0,Y 538.046,Z 720.273,A -85,B 0,C 180,E1 -4075.673,E2 -4075.673} C_VEL
LIN {X 0,Y 538.045,Z 720.272,A -85,B 0,C 180,E1 -4078.05,E2 -4078.05} C_VEL
LIN {X 0,Y 538.022,Z 720.27,A -85,B 0,C 180,E1 -4080.627,E2 -4080.627} C_VEL
LIN {X 0,Y 538.046,Z 720.279,A -85,B 0,C 180,E1 -4083.283,E2 -4083.283} C_VEL
LIN {X 0,Y 538.029,Z 720.273,A -85,B 0,C 180,E1 -4086.002,E2 -4086.002} C_VEL
LIN {X 0,Y 538.02,Z 720.275,A -85,B 0,C 180,E1 -4088.83,E2 -4088.83} C_VEL
LIN {X 0,Y 538.04,Z 720.273,A -85,B 0,C 180,E1 -4091.88,E2 -4091.88} C_VEL
LIN {X 0,Y 538.033,Z 720.275,A -85,B 0,C 180,E1 -4095.141,E2 -4095.141} C_VEL
LIN {X 0,Y 538.042,Z 720.267,A -85,B 0,C 180,E1 -4098.228,E2 -4098.228} C_VEL
LIN {X 0,Y 538.061,Z 720.254,A -85,B 0,C 180,E1 -4100.412,E2 -4100.412} C_VEL
LIN {X 0,Y 538.031,Z 720.267,A -85,B 0,C 180,E1 -4103.068,E2 -4103.068} C_VEL
LIN {X 0,Y 538.03,Z 720.282,A -85,B 0,C 180,E1 -4105.828,E2 -4105.828} C_VEL
LIN {X 0,Y 538.012,Z 720.275,A -85,B 0,C 180,E1 -4108.499,E2 -4108.499} C_VEL
LIN {X 0,Y 538.061,Z 720.265,A -85,B 0,C 180,E1 -4111.1,E2 -4111.1} C_VEL
LIN {X 0,Y 538.044,Z 720.275,A -85,B 0,C 180,E1 -4113.634,E2 -4113.634} C_VEL
LIN {X 0,Y 538.025,Z 720.279,A -85,B 0,C 180,E1 -4116.118,E2 -4116.118} C_VEL
LIN {X 0,Y 538.042,Z 720.267,A -85,B 0,C 180,E1 -4119.349,E2 -4119.349} C_VEL
LIN {X 0,Y 538.076,Z 720.271,A -85,B 0,C 180,E1 -4122.518,E2 -4122.518} C_VEL
LIN {X 0,Y 538.066,Z 720.268,A -85,B 0,C 180,E1 -4125.631,E2 -4125.631} C_VEL
LIN {X 0,Y 538.08,Z 720.266,A -85,B 0,C 180,E1 -4128.702,E2 -4128.702} C_VEL
LIN {X 0,Y 538.089,Z 720.266,A -85,B 0,C 180,E1 -4131.74,E2 -4131.74} C_VEL
LIN {X 0,Y 538.163,Z 720.258,A -85,B 0,C 180,E1 -4134.755,E2 -4134.755} C_VEL
LIN {X 0,Y 538.17,Z 720.249,A -85,B 0,C 180,E1 -4137.755,E2 -4137.755} C_VEL
LIN {X 0,Y 538.186,Z 720.259,A -85,B 0,C 180,E1 -4140.748,E2 -4140.748} C_VEL
LIN {X 0,Y 538.142,Z 720.261,A -85,B 0,C 180,E1 -4142.995,E2 -4142.995} C_VEL
LIN {X 0,Y 538.123,Z 720.259,A -85,B 0,C 180,E1 -4145.997,E2 -4145.997} C_VEL
LIN {X 0,Y 538.064,Z 720.271,A -85,B 0,C 180,E1 -4149.018,E2 -4149.018} C_VEL
LIN {X 0,Y 538.086,Z 720.266,A -85,B 0,C 180,E1 -4152.063,E2 -4152.063} C_VEL
LIN {X 0,Y 538.048,Z 720.272,A -85,B 0,C 180,E1 -4155.144,E2 -4155.144} C_VEL
LIN {X 0,Y 538.028,Z 720.269,A -85,B 0,C 180,E1 -4158.27,E2 -4158.27} C_VEL
LIN {X 0,Y 538.04,Z 720.275,A -85,B 0,C 180,E1 -4160.651,E2 -4160.651} C_VEL
LIN {X 0,Y 538.004,Z 720.274,A -85,B 0,C 180,E1 -4163.888,E2 -4163.888} C_VEL
LIN {X 0,Y 538.043,Z 720.267,A -85,B 0,C 180,E1 -4166.367,E2 -4166.367} C_VEL
LIN {X 0,Y 538.032,Z 720.278,A -85,B 0,C 180,E1 -4168.933,E2 -4168.933} C_VEL
LIN {X 0,Y 538.012,Z 720.273,A -85,B 0,C 180,E1 -4171.887,E2 -4171.887} C_VEL
LIN {X 0,Y 538.011,Z 720.274,A -85,B 0,C 180,E1 -4174.617,E2 -4174.617} C_VEL
LIN {X 0,Y 538.005,Z 720.284,A -85,B 0,C 180,E1 -4177.17,E2 -4177.17} C_VEL
LIN {X 0,Y 538.017,Z 720.269,A -85,B 0,C 180,E1 -4180.26,E2 -4180.26} C_VEL
LIN {X 0,Y 537.367,Z 720.354,A -85,B 0,C 180,E1 -4180.885,E2 -4180.885} C_VEL
LIN {X 0,Y 534.51,Z 720.712,A -85,B 0,C 180,E1 -4181.9,E2 -4181.9} C_VEL
LIN {X 0,Y 532.081,Z 721.016,A -85,B 0,C 180,E1 -4182.717,E2 -4182.717} C_VEL
LIN {X 0,Y 531.033,Z 721.143,A -85,B 0,C 180,E1 -4183.348,E2 -4183.348} C_VEL
LIN {X 0,Y 530.946,Z 721.152,A -85,B 0,C 180,E1 -4183.562,E2 -4183.562} C_VEL
LIN {X 0,Y 530.955,Z 721.153,A -85,B 0,C 180,E1 -4186.504,E2 -4186.504} C_VEL
LIN {X 0,Y 530.985,Z 721.152,A -85,B 0,C 180,E1 -4188.977,E2 -4188.977} C_VEL
LIN {X 0,Y 530.958,Z 721.155,A -85,B 0,C 180,E1 -4191.529,E2 -4191.529} C_VEL
LIN {X 0,Y 530.955,Z 721.155,A -85,B 0,C 180,E1 -4194.38,E2 -4194.38} C_VEL
LIN {X 0,Y 530.968,Z 721.154,A -85,B 0,C 180,E1 -4197.133,E2 -4197.133} C_VEL
LIN {X 0,Y 530.962,Z 721.162,A -85,B 0,C 180,E1 -4199.803,E2 -4199.803} C_VEL
LIN {X 0,Y 530.974,Z 721.153,A -85,B 0,C 180,E1 -4202.476,E2 -4202.476} C_VEL
LIN {X 0,Y 530.969,Z 721.153,A -85,B 0,C 180,E1 -4204.941,E2 -4204.941} C_VEL
LIN {X 0,Y 530.979,Z 721.161,A -85,B 0,C 180,E1 -4207.898,E2 -4207.898} C_VEL
LIN {X 0,Y 531.009,Z 721.154,A -85,B 0,C 180,E1 -4210.678,E2 -4210.678} C_VEL
LIN {X 0,Y 531.098,Z 721.35,A -85,B 0,C 180,E1 -4211.483,E2 -4211.483} C_VEL
LIN {X 0,Y 531.129,Z 728.157,A -85,B 0,C 180,E1 -4213.076,E2 -4213.076} C_VEL
LIN {X 0,Y 530.921,Z 740.281,A -85,B 0,C 180,E1 -4215.825,E2 -4215.825} C_VEL
LIN {X 0,Y 530.788,Z 751.447,A -85,B 0,C 180,E1 -4218.287,E2 -4218.287} C_VEL
LIN {X 0,Y 531.897,Z 759.435,A -85,B 0,C 180,E1 -4218.444,E2 -4218.444} C_VEL
LIN {X 0,Y 531.699,Z 826.319,A -85,B 0,C 180,E1 -4219.36,E2 -4219.36} C_VEL
LIN {X 0,Y 531.629,Z 835.534,A -85,B 0,C 180,E1 -4219.575,E2 -4219.575} C_VEL
LIN {X 0,Y 531.533,Z 845.187,A -85,B 0,C 180,E1 -4219.91,E2 -4219.91} C_VEL
LIN {X 0,Y 531.396,Z 855.261,A -85,B 0,C 180,E1 -4220.388,E2 -4220.388} C_VEL
LIN {X 0,Y 531.22,Z 865.725,A -85,B 0,C 180,E1 -4221.057,E2 -4221.057} C_VEL
LIN {X 0,Y 530.993,Z 873.898,A -85,B 0,C 180,E1 -4221.724,E2 -4221.724} C_VEL
LIN {X 0,Y 530.842,Z 880.639,A -85,B 0,C 180,E1 -4222.392,E2 -4222.392} C_VEL
LIN {X 0,Y 530.742,Z 887.982,A -85,B 0,C 180,E1 -4223.284,E2 -4223.284} C_VEL
LIN {X 0,Y 530.71,Z 893.506,A -85,B 0,C 180,E1 -4224.109,E2 -4224.109} C_VEL
LIN {X 0,Y 530.506,Z 898.674,A -85,B 0,C 180,E1 -4225.06,E2 -4225.06} C_VEL
LIN {X 0,Y 530.525,Z 903.465,A -85,B 0,C 180,E1 -4226.202,E2 -4226.202} C_VEL
LIN {X 0,Y 530.47,Z 905.804,A -85,B 0,C 180,E1 -4226.962,E2 -4226.962} C_VEL
LIN {X 0,Y 530.412,Z 907.589,A -85,B 0,C 180,E1 -4227.722,E2 -4227.722} C_VEL
LIN {X 0,Y 530.359,Z 908.875,A -85,B 0,C 180,E1 -4228.481,E2 -4228.481} C_VEL
LIN {X 0,Y 530.34,Z 909.69,A -85,B 0,C 180,E1 -4229.241,E2 -4229.241} C_VEL
LIN {X 0,Y 530.341,Z 909.997,A -85,B 0,C 180,E1 -4230,E2 -4230} C_VEL
LIN {X 0,Y 530.341,Z 909.727,A -85,B 0,C 180,E1 -4230.759,E2 -4230.759} C_VEL
LIN {X 0,Y 530.36,Z 908.989,A -85,B 0,C 180,E1 -4231.519,E2 -4231.519} C_VEL
LIN {X 0,Y 530.413,Z 907.781,A -85,B 0,C 180,E1 -4232.278,E2 -4232.278} C_VEL
LIN {X 0,Y 530.494,Z 904.925,A -85,B 0,C 180,E1 -4233.418,E2 -4233.418} C_VEL
LIN {X 0,Y 530.545,Z 902.33,A -85,B 0,C 180,E1 -4234.178,E2 -4234.178} C_VEL
LIN {X 0,Y 530.541,Z 897.214,A -85,B 0,C 180,E1 -4235.321,E2 -4235.321} C_VEL
LIN {X 0,Y 530.728,Z 891.746,A -85,B 0,C 180,E1 -4236.266,E2 -4236.266} C_VEL
LIN {X 0,Y 530.791,Z 884.815,A -85,B 0,C 180,E1 -4237.226,E2 -4237.226} C_VEL
LIN {X 0,Y 530.957,Z 875.881,A -85,B 0,C 180,E1 -4238.181,E2 -4238.181} C_VEL
LIN {X 0,Y 531.139,Z 868.114,A -85,B 0,C 180,E1 -4238.848,E2 -4238.848} C_VEL
LIN {X 0,Y 531.26,Z 859.925,A -85,B 0,C 180,E1 -4239.422,E2 -4239.422} C_VEL
LIN {X 0,Y 531.445,Z 849.52,A -85,B 0,C 180,E1 -4239.995,E2 -4239.995} C_VEL
LIN {X 0,Y 531.64,Z 837.819,A -85,B 0,C 180,E1 -4240.449,E2 -4240.449} C_VEL
LIN {X 0,Y 531.747,Z 828.579,A -85,B 0,C 180,E1 -4240.687,E2 -4240.687} C_VEL
LIN {X 0,Y 531.807,Z 802.142,A -85,B 0,C 180,E1 -4241.072,E2 -4241.072} C_VEL
LIN {X 0,Y 531.742,Z 757.949,A -85,B 0,C 180,E1 -4241.669,E2 -4241.669} C_VEL
LIN {X 0,Y 530.801,Z 751.838,A -85,B 0,C 180,E1 -4241.797,E2 -4241.797} C_VEL
LIN {X 0,Y 530.754,Z 750.928,A -85,B 0,C 180,E1 -4241.892,E2 -4241.892} C_VEL
LIN {X 0,Y 531.013,Z 737.238,A -85,B 0,C 180,E1 -4244.948,E2 -4244.948} C_VEL
LIN {X 0,Y 531.176,Z 723.392,A -85,B 0,C 180,E1 -4248.115,E2 -4248.115} C_VEL
LIN {X 0,Y 531.053,Z 721.229,A -85,B 0,C 180,E1 -4248.669,E2 -4248.669} C_VEL
LIN {X 0,Y 531,Z 721.15,A -85,B 0,C 180,E1 -4250.938,E2 -4250.938} C_VEL
LIN {X 0,Y 530.955,Z 721.162,A -85,B 0,C 180,E1 -4254.226,E2 -4254.226} C_VEL
LIN {X 0,Y 530.966,Z 721.156,A -85,B 0,C 180,E1 -4256.746,E2 -4256.746} C_VEL
LIN {X 0,Y 530.981,Z 721.151,A -85,B 0,C 180,E1 -4259.323,E2 -4259.323} C_VEL
LIN {X 0,Y 530.966,Z 721.155,A -85,B 0,C 180,E1 -4262.1,E2 -4262.1} C_VEL
LIN {X 0,Y 530.969,Z 721.157,A -85,B 0,C 180,E1 -4264.851,E2 -4264.851} C_VEL
LIN {X 0,Y 530.966,Z 721.149,A -85,B 0,C 180,E1 -4267.508,E2 -4267.508} C_VEL
LIN {X 0,Y 530.979,Z 721.155,A -85,B 0,C 180,E1 -4270.433,E2 -4270.433} C_VEL
LIN {X 0,Y 530.962,Z 721.154,A -85,B 0,C 180,E1 -4273.281,E2 -4273.281} C_VEL
LIN {X 0,Y 530.977,Z 721.146,A -85,B 0,C 180,E1 -4275.622,E2 -4275.622} C_VEL
LIN {X 0,Y 530.994,Z 721.143,A -85,B 0,C 180,E1 -4278.564,E2 -4278.564} C_VEL
LIN {X 0,Y 530.956,Z 721.153,A -85,B 0,C 180,E1 -4281.529,E2 -4281.529} C_VEL
LIN {X 0,Y 530.955,Z 721.157,A -85,B 0,C 180,E1 -4284.38,E2 -4284.38} C_VEL
LIN {X 0,Y 530.968,Z 721.156,A -85,B 0,C 180,E1 -4287.133,E2 -4287.133} C_VEL
LIN {X 0,Y 530.962,Z 721.153,A -85,B 0,C 180,E1 -4289.802,E2 -4289.802} C_VEL
LIN {X 0,Y 531.013,Z 721.148,A -85,B 0,C 180,E1 -4292.468,E2 -4292.468} C_VEL
LIN {X 0,Y 531.001,Z 721.151,A -85,B 0,C 180,E1 -4294.942,E2 -4294.942} C_VEL
LIN {X 0,Y 530.973,Z 721.152,A -85,B 0,C 180,E1 -4298.247,E2 -4298.247} C_VEL
LIN {X 0,Y 530.995,Z 721.151,A -85,B 0,C 180,E1 -4300.677,E2 -4300.677} C_VEL
LIN {X 0,Y 530.978,Z 721.153,A -85,B 0,C 180,E1 -4303.071,E2 -4303.071} C_VEL
LIN {X 0,Y 531.043,Z 721.149,A -85,B 0,C 180,E1 -4305.436,E2 -4305.436} C_VEL
LIN {X 0,Y 531.04,Z 721.144,A -85,B 0,C 180,E1 -4308.55,E2 -4308.55} C_VEL
LIN {X 0,Y 531.055,Z 721.139,A -85,B 0,C 180,E1 -4311.629,E2 -4311.629} C_VEL
LIN {X 0,Y 531.125,Z 721.13,A -85,B 0,C 180,E1 -4314.685,E2 -4314.685} C_VEL
LIN {X 0,Y 531.144,Z 721.136,A -85,B 0,C 180,E1 -4317.725,E2 -4317.725} C_VEL
LIN {X 0,Y 531.155,Z 721.126,A -85,B 0,C 180,E1 -4320.758,E2 -4320.758} C_VEL
LIN {X 0,Y 531.108,Z 721.129,A -85,B 0,C 180,E1 -4323.034,E2 -4323.034} C_VEL
LIN {X 0,Y 531.083,Z 721.141,A -85,B 0,C 180,E1 -4326.077,E2 -4326.077} C_VEL
LIN {X 0,Y 531.034,Z 721.145,A -85,B 0,C 180,E1 -4329.138,E2 -4329.138} C_VEL
LIN {X 0,Y 531.043,Z 721.14,A -85,B 0,C 180,E1 -4332.225,E2 -4332.225} C_VEL
LIN {X 0,Y 530.999,Z 721.149,A -85,B 0,C 180,E1 -4335.35,E2 -4335.35} C_VEL
LIN {X 0,Y 531.019,Z 721.153,A -85,B 0,C 180,E1 -4337.722,E2 -4337.722} C_VEL
LIN {X 0,Y 531.002,Z 721.142,A -85,B 0,C 180,E1 -4340.938,E2 -4340.938} C_VEL
LIN {X 0,Y 530.982,Z 721.157,A -85,B 0,C 180,E1 -4344.224,E2 -4344.224} C_VEL
LIN {X 0,Y 531.008,Z 721.147,A -85,B 0,C 180,E1 -4346.743,E2 -4346.743} C_VEL
LIN {X 0,Y 530.984,Z 721.146,A -85,B 0,C 180,E1 -4349.322,E2 -4349.322} C_VEL
LIN {X 0,Y 530.972,Z 721.159,A -85,B 0,C 180,E1 -4352.101,E2 -4352.101} C_VEL
LIN {X 0,Y 530.991,Z 721.149,A -85,B 0,C 180,E1 -4354.854,E2 -4354.854} C_VEL
LIN {X 0,Y 530.968,Z 721.146,A -85,B 0,C 180,E1 -4357.507,E2 -4357.507} C_VEL
LIN {X 0,Y 531.028,Z 721.142,A -85,B 0,C 180,E1 -4360.429,E2 -4360.429} C_VEL
LIN {X 0,Y 530.966,Z 721.152,A -85,B 0,C 180,E1 -4363.494,E2 -4363.494} C_VEL
LIN {X 0,Y 530.961,Z 721.159,A -85,B 0,C 180,E1 -4366.505,E2 -4366.505} C_VEL
LIN {X 0,Y 530.991,Z 721.149,A -85,B 0,C 180,E1 -4368.976,E2 -4368.976} C_VEL
LIN {X 0,Y 530.962,Z 721.153,A -85,B 0,C 180,E1 -4371.53,E2 -4371.53} C_VEL
LIN {X 0,Y 530.984,Z 721.154,A -85,B 0,C 180,E1 -4374.382,E2 -4374.382} C_VEL
LIN {X 0,Y 530.974,Z 721.153,A -85,B 0,C 180,E1 -4377.134,E2 -4377.134} C_VEL
LIN {X 0,Y 530.971,Z 721.147,A -85,B 0,C 180,E1 -4379.803,E2 -4379.803} C_VEL
LIN {X 0,Y 531.016,Z 721.153,A -85,B 0,C 180,E1 -4382.467,E2 -4382.467} C_VEL
LIN {X 0,Y 530.996,Z 721.156,A -85,B 0,C 180,E1 -4384.942,E2 -4384.942} C_VEL
LIN {X 0,Y 531.03,Z 721.277,A -85,B 0,C 180,E1 -4387.521,E2 -4387.521} C_VEL
LIN {X 0,Y 531.86,Z 727.309,A -85,B 0,C 180,E1 -4388.692,E2 -4388.692} C_VEL
LIN {X 0,Y 531.582,Z 743.828,A -85,B 0,C 180,E1 -4391.72,E2 -4391.72} C_VEL
LIN {X 0,Y 531.251,Z 760.018,A -85,B 0,C 180,E1 -4394.658,E2 -4394.658} C_VEL
LIN {X 0,Y 530.937,Z 777.321,A -85,B 0,C 180,E1 -4397.773,E2 -4397.773} C_VEL
LIN {X 0,Y 530.938,Z 780.102,A -85,B 0,C 180,E1 -4398.224,E2 -4398.224} C_VEL
LIN {X 0,Y 531.928,Z 788.986,A -85,B 0,C 180,E1 -4398.394,E2 -4398.394} C_VEL
LIN {X 0,Y 531.768,Z 856.138,A -85,B 0,C 180,E1 -4399.313,E2 -4399.313} C_VEL
LIN {X 0,Y 531.644,Z 865.41,A -85,B 0,C 180,E1 -4399.527,E2 -4399.527} C_VEL
LIN {X 0,Y 531.548,Z 873.884,A -85,B 0,C 180,E1 -4399.814,E2 -4399.814} C_VEL
LIN {X 0,Y 531.41,Z 882.39,A -85,B 0,C 180,E1 -4400.196,E2 -4400.196} C_VEL
LIN {X 0,Y 531.242,Z 890.724,A -85,B 0,C 180,E1 -4400.674,E2 -4400.674} C_VEL
LIN {X 0,Y 531.109,Z 898.763,A -85,B 0,C 180,E1 -4401.247,E2 -4401.247} C_VEL
LIN {X 0,Y 530.93,Z 906.415,A -85,B 0,C 180,E1 -4401.915,E2 -4401.915} C_VEL
LIN {X 0,Y 530.809,Z 914.435,A -85,B 0,C 180,E1 -4402.774,E2 -4402.774} C_VEL
LIN {X 0,Y 530.728,Z 921.45,A -85,B 0,C 180,E1 -4403.73,E2 -4403.73} C_VEL
LIN {X 0,Y 530.542,Z 926.989,A -85,B 0,C 180,E1 -4404.679,E2 -4404.679} C_VEL
LIN {X 0,Y 530.547,Z 932.149,A -85,B 0,C 180,E1 -4405.822,E2 -4405.822} C_VEL
LIN {X 0,Y 530.469,Z 935.937,A -85,B 0,C 180,E1 -4406.962,E2 -4406.962} C_VEL
LIN {X 0,Y 530.41,Z 937.682,A -85,B 0,C 180,E1 -4407.722,E2 -4407.722} C_VEL
LIN {X 0,Y 530.359,Z 938.931,A -85,B 0,C 180,E1 -4408.481,E2 -4408.481} C_VEL
LIN {X 0,Y 530.342,Z 939.707,A -85,B 0,C 180,E1 -4409.241,E2 -4409.241} C_VEL
LIN {X 0,Y 530.34,Z 940,A -85,B 0,C 180,E1 -4410,E2 -4410} C_VEL
LIN {X 0,Y 530.342,Z 939.707,A -85,B 0,C 180,E1 -4410.759,E2 -4410.759} C_VEL
LIN {X 0,Y 530.359,Z 938.93,A -85,B 0,C 180,E1 -4411.519,E2 -4411.519} C_VEL
LIN {X 0,Y 530.41,Z 937.681,A -85,B 0,C 180,E1 -4412.278,E2 -4412.278} C_VEL
LIN {X 0,Y 530.495,Z 934.787,A -85,B 0,C 180,E1 -4413.418,E2 -4413.418} C_VEL
LIN {X 0,Y 530.547,Z 932.149,A -85,B 0,C 180,E1 -4414.178,E2 -4414.178} C_VEL
LIN {X 0,Y 530.542,Z 926.986,A -85,B 0,C 180,E1 -4415.321,E2 -4415.321} C_VEL
LIN {X 0,Y 530.729,Z 921.441,A -85,B 0,C 180,E1 -4416.27,E2 -4416.27} C_VEL
LIN {X 0,Y 530.794,Z 914.435,A -85,B 0,C 180,E1 -4417.226,E2 -4417.226} C_VEL
LIN {X 0,Y 530.93,Z 906.421,A -85,B 0,C 180,E1 -4418.085,E2 -4418.085} C_VEL
LIN {X 0,Y 531.109,Z 898.767,A -85,B 0,C 180,E1 -4418.753,E2 -4418.753} C_VEL
LIN {X 0,Y 531.242,Z 890.724,A -85,B 0,C 180,E1 -4419.326,E2 -4419.326} C_VEL
LIN {X 0,Y 531.41,Z 882.392,A -85,B 0,C 180,E1 -4419.804,E2 -4419.804} C_VEL
LIN {X 0,Y 531.548,Z 873.887,A -85,B 0,C 180,E1 -4420.186,E2 -4420.186} C_VEL
LIN {X 0,Y 531.638,Z 863.749,A -85,B 0,C 180,E1 -4420.521,E2 -4420.521} C_VEL
LIN {X 0,Y 531.816,Z 852.057,A -85,B 0,C 180,E1 -4420.758,E2 -4420.758} C_VEL
LIN {X 0,Y 531.773,Z 786.763,A -85,B 0,C 180,E1 -4421.64,E2 -4421.64} C_VEL
LIN {X 0,Y 530.927,Z 780.15,A -85,B 0,C 180,E1 -4421.773,E2 -4421.773} C_VEL
LIN {X 0,Y 530.992,Z 772.996,A -85,B 0,C 180,E1 -4423.003,E2 -4423.003} C_VEL
LIN {X 0,Y 531.259,Z 757.856,A -85,B 0,C 180,E1 -4425.735,E2 -4425.735} C_VEL
LIN {X 0,Y 531.569,Z 742.625,A -85,B 0,C 180,E1 -4428.5,E2 -4428.5} C_VEL
LIN {X 0,Y 531.858,Z 727.309,A -85,B 0,C 180,E1 -4431.308,E2 -4431.308} C_VEL
LIN {X 0,Y 531.004,Z 721.212,A -85,B 0,C 180,E1 -4432.511,E2 -4432.511} C_VEL
LIN {X 0,Y 531.015,Z 721.147,A -85,B 0,C 180,E1 -4435.897,E2 -4435.897} C_VEL
LIN {X 0,Y 531,Z 721.15,A -85,B 0,C 180,E1 -4438.455,E2 -4438.455} C_VEL
LIN {X 0,Y 530.966,Z 721.152,A -85,B 0,C 180,E1 -4441.079,E2 -4441.079} C_VEL
LIN {X 0,Y 530.992,Z 721.154,A -85,B 0,C 180,E1 -4443.772,E2 -4443.772} C_VEL
LIN {X 0,Y 530.97,Z 721.15,A -85,B 0,C 180,E1 -4446.557,E2 -4446.557} C_VEL
LIN {X 0,Y 530.988,Z 721.15,A -85,B 0,C 180,E1 -4449.855,E2 -4449.855} C_VEL
LIN {X 0,Y 530.982,Z 721.147,A -85,B 0,C 180,E1 -4452.456,E2 -4452.456} C_VEL
LIN {X 0,Y 530.989,Z 721.159,A -85,B 0,C 180,E1 -4455.621,E2 -4455.621} C_VEL
LIN {X 0,Y 531.009,Z 721.141,A -85,B 0,C 180,E1 -4458.566,E2 -4458.566} C_VEL
LIN {X 0,Y 530.97,Z 721.139,A -85,B 0,C 180,E1 -4461.346,E2 -4461.346} C_VEL
LIN {X 0,Y 530.984,Z 721.15,A -85,B 0,C 180,E1 -4464.382,E2 -4464.382} C_VEL
LIN {X 0,Y 530.972,Z 721.153,A -85,B 0,C 180,E1 -4467.134,E2 -4467.134} C_VEL
LIN {X 0,Y 530.972,Z 721.158,A -85,B 0,C 180,E1 -4469.803,E2 -4469.803} C_VEL
LIN {X 0,Y 531.017,Z 721.148,A -85,B 0,C 180,E1 -4472.467,E2 -4472.467} C_VEL
LIN {X 0,Y 531.008,Z 721.147,A -85,B 0,C 180,E1 -4474.943,E2 -4474.943} C_VEL
LIN {X 0,Y 530.974,Z 721.153,A -85,B 0,C 180,E1 -4478.247,E2 -4478.247} C_VEL
LIN {X 0,Y 530.999,Z 721.149,A -85,B 0,C 180,E1 -4480.678,E2 -4480.678} C_VEL
LIN {X 0,Y 530.994,Z 721.149,A -85,B 0,C 180,E1 -4483.071,E2 -4483.071} C_VEL
LIN {X 0,Y 531.022,Z 721.144,A -85,B 0,C 180,E1 -4485.436,E2 -4485.436} C_VEL
LIN {X 0,Y 531.039,Z 721.145,A -85,B 0,C 180,E1 -4488.55,E2 -4488.55} C_VEL
LIN {X 0,Y 531.059,Z 721.141,A -85,B 0,C 180,E1 -4491.63,E2 -4491.63} C_VEL
LIN {X 0,Y 531.123,Z 721.136,A -85,B 0,C 180,E1 -4494.685,E2 -4494.685} C_VEL
LIN {X 0,Y 531.142,Z 721.123,A -85,B 0,C 180,E1 -4497.725,E2 -4497.725} C_VEL
LIN {X 0,Y 531.156,Z 721.134,A -85,B 0,C 180,E1 -4500.758,E2 -4500.758} C_VEL
LIN {X 0,Y 531.109,Z 721.137,A -85,B 0,C 180,E1 -4503.034,E2 -4503.034} C_VEL
LIN {X 0,Y 531.078,Z 721.137,A -85,B 0,C 180,E1 -4506.077,E2 -4506.077} C_VEL
LIN {X 0,Y 531.055,Z 721.138,A -85,B 0,C 180,E1 -4508.371,E2 -4508.371} C_VEL
LIN {X 0,Y 531.054,Z 721.141,A -85,B 0,C 180,E1 -4511.672,E2 -4511.672} C_VEL
LIN {X 0,Y 531.033,Z 721.148,A -85,B 0,C 180,E1 -4514.956,E2 -4514.956} C_VEL
LIN {X 0,Y 530.983,Z 721.145,A -85,B 0,C 180,E1 -4517.724,E2 -4517.724} C_VEL
LIN {X 0,Y 531.027,Z 721.144,A -85,B 0,C 180,E1 -4520.127,E2 -4520.127} C_VEL
LIN {X 0,Y 530.947,Z 721.158,A -85,B 0,C 180,E1 -4522.573,E2 -4522.573} C_VEL
LIN {X 0,Y 530.991,Z 721.153,A -85,B 0,C 180,E1 -4525.058,E2 -4525.058} C_VEL
LIN {X 0,Y 531.015,Z 721.147,A -85,B 0,C 180,E1 -4527.596,E2 -4527.596} C_VEL
LIN {X 0,Y 530.968,Z 721.155,A -85,B 0,C 180,E1 -4530.644,E2 -4530.644} C_VEL
LIN {X 0,Y 530.964,Z 721.155,A -85,B 0,C 180,E1 -4533.5,E2 -4533.5} C_VEL
LIN {X 0,Y 530.946,Z 721.155,A -85,B 0,C 180,E1 -4536.153,E2 -4536.153} C_VEL
LIN {X 0,Y 530.965,Z 721.153,A -85,B 0,C 180,E1 -4538.653,E2 -4538.653} C_VEL
LIN {X 0,Y 530.995,Z 721.144,A -85,B 0,C 180,E1 -4541.436,E2 -4541.436} C_VEL
LIN {X 0,Y 530.946,Z 721.152,A -85,B 0,C 180,E1 -4543.562,E2 -4543.562} C_VEL
LIN {X 0,Y 530.277,Z 721.234,A -85,B 0,C 180,E1 -4544.195,E2 -4544.195} C_VEL
LIN {X 0,Y 527.433,Z 721.593,A -85,B 0,C 180,E1 -4545.224,E2 -4545.224} C_VEL
LIN {X 0,Y 525.032,Z 721.893,A -85,B 0,C 180,E1 -4546.053,E2 -4546.053} C_VEL
LIN {X 0,Y 524,Z 722.021,A -85,B 0,C 180,E1 -4546.692,E2 -4546.692} C_VEL
LIN {X 0,Y 523.916,Z 722.032,A -85,B 0,C 180,E1 -4546.909,E2 -4546.909} C_VEL
LIN {X 0,Y 523.95,Z 722.026,A -85,B 0,C 180,E1 -4549.921,E2 -4549.921} C_VEL
LIN {X 0,Y 523.908,Z 722.028,A -85,B 0,C 180,E1 -4552.868,E2 -4552.868} C_VEL
LIN {X 0,Y 523.921,Z 722.039,A -85,B 0,C 180,E1 -4555.709,E2 -4555.709} C_VEL
LIN {X 0,Y 523.921,Z 722.027,A -85,B 0,C 180,E1 -4558.456,E2 -4558.456} C_VEL
LIN {X 0,Y 523.928,Z 722.031,A -85,B 0,C 180,E1 -4561.125,E2 -4561.125} C_VEL
LIN {X 0,Y 523.928,Z 722.037,A -85,B 0,C 180,E1 -4563.993,E2 -4563.993} C_VEL
LIN {X 0,Y 523.911,Z 722.034,A -85,B 0,C 180,E1 -4566.269,E2 -4566.269} C_VEL
LIN {X 0,Y 523.947,Z 722.029,A -85,B 0,C 180,E1 -4568.767,E2 -4568.767} C_VEL
LIN {X 0,Y 524.06,Z 722.153,A -85,B 0,C 180,E1 -4571.377,E2 -4571.377} C_VEL
LIN {X 0,Y 524.142,Z 728.305,A -85,B 0,C 180,E1 -4572.843,E2 -4572.843} C_VEL
LIN {X 0,Y 523.893,Z 740.384,A -85,B 0,C 180,E1 -4575.63,E2 -4575.63} C_VEL
LIN {X 0,Y 523.725,Z 751.413,A -85,B 0,C 180,E1 -4578.104,E2 -4578.104} C_VEL
LIN {X 0,Y 524.027,Z 753.621,A -85,B 0,C 180,E1 -4578.188,E2 -4578.188} C_VEL
LIN {X 0,Y 524.968,Z 760.799,A -85,B 0,C 180,E1 -4578.308,E2 -4578.308} C_VEL
LIN {X 0,Y 524.735,Z 826.352,A -85,B 0,C 180,E1 -4579.217,E2 -4579.217} C_VEL
LIN {X 0,Y 524.669,Z 835.554,A -85,B 0,C 180,E1 -4579.435,E2 -4579.435} C_VEL
LIN {X 0,Y 524.534,Z 845.201,A -85,B 0,C 180,E1 -4579.774,E2 -4579.774} C_VEL
LIN {X 0,Y 524.399,Z 855.276,A -85,B 0,C 180,E1 -4580.259,E2 -4580.259} C_VEL
LIN {X 0,Y 524.2,Z 865.73,A -85,B 0,C 180,E1 -4580.936,E2 -4580.936} C_VEL
LIN {X 0,Y 523.95,Z 873.903,A -85,B 0,C 180,E1 -4581.612,E2 -4581.612} C_VEL
LIN {X 0,Y 523.797,Z 880.643,A -85,B 0,C 180,E1 -4582.289,E2 -4582.289} C_VEL
LIN {X 0,Y 523.704,Z 887.027,A -85,B 0,C 180,E1 -4583.063,E2 -4583.063} C_VEL
LIN {X 0,Y 523.656,Z 892.335,A -85,B 0,C 180,E1 -4583.836,E2 -4583.836} C_VEL
LIN {X 0,Y 523.488,Z 896.766,A -85,B 0,C 180,E1 -4584.608,E2 -4584.608} C_VEL
LIN {X 0,Y 523.416,Z 900.455,A -85,B 0,C 180,E1 -4585.379,E2 -4585.379} C_VEL
LIN {X 0,Y 523.454,Z 903.468,A -85,B 0,C 180,E1 -4586.151,E2 -4586.151} C_VEL
LIN {X 0,Y 523.381,Z 905.807,A -85,B 0,C 180,E1 -4586.921,E2 -4586.921} C_VEL
LIN {X 0,Y 523.336,Z 907.589,A -85,B 0,C 180,E1 -4587.691,E2 -4587.691} C_VEL
LIN {X 0,Y 523.273,Z 908.875,A -85,B 0,C 180,E1 -4588.461,E2 -4588.461} C_VEL
LIN {X 0,Y 523.246,Z 909.689,A -85,B 0,C 180,E1 -4589.23,E2 -4589.23} C_VEL
LIN {X 0,Y 523.244,Z 909.997,A -85,B 0,C 180,E1 -4590,E2 -4590} C_VEL
LIN {X 0,Y 523.247,Z 909.727,A -85,B 0,C 180,E1 -4590.77,E2 -4590.77} C_VEL
LIN {X 0,Y 523.274,Z 908.988,A -85,B 0,C 180,E1 -4591.539,E2 -4591.539} C_VEL
LIN {X 0,Y 523.337,Z 907.779,A -85,B 0,C 180,E1 -4592.309,E2 -4592.309} C_VEL
LIN {X 0,Y 523.406,Z 904.923,A -85,B 0,C 180,E1 -4593.464,E2 -4593.464} C_VEL
LIN {X 0,Y 523.468,Z 902.328,A -85,B 0,C 180,E1 -4594.235,E2 -4594.235} C_VEL
LIN {X 0,Y 523.484,Z 897.211,A -85,B 0,C 180,E1 -4595.393,E2 -4595.393} C_VEL
LIN {X 0,Y 523.642,Z 892.882,A -85,B 0,C 180,E1 -4596.164,E2 -4596.164} C_VEL
LIN {X 0,Y 523.701,Z 886.266,A -85,B 0,C 180,E1 -4597.131,E2 -4597.131} C_VEL
LIN {X 0,Y 523.86,Z 877.912,A -85,B 0,C 180,E1 -4598.098,E2 -4598.098} C_VEL
LIN {X 0,Y 524.094,Z 869.336,A -85,B 0,C 180,E1 -4598.871,E2 -4598.871} C_VEL
LIN {X 0,Y 524.232,Z 861.419,A -85,B 0,C 180,E1 -4599.452,E2 -4599.452} C_VEL
LIN {X 0,Y 524.4,Z 853.259,A -85,B 0,C 180,E1 -4599.936,E2 -4599.936} C_VEL
LIN {X 0,Y 524.541,Z 845.014,A -85,B 0,C 180,E1 -4600.323,E2 -4600.323} C_VEL
LIN {X 0,Y 524.662,Z 836.129,A -85,B 0,C 180,E1 -4600.638,E2 -4600.638} C_VEL
LIN {X 0,Y 524.802,Z 827.245,A -85,B 0,C 180,E1 -4600.855,E2 -4600.855} C_VEL
LIN {X 0,Y 524.812,Z 758.885,A -85,B 0,C 180,E1 -4601.812,E2 -4601.812} C_VEL
LIN {X 0,Y 523.778,Z 752.239,A -85,B 0,C 180,E1 -4601.938,E2 -4601.938} C_VEL
LIN {X 0,Y 523.701,Z 750.918,A -85,B 0,C 180,E1 -4602.055,E2 -4602.055} C_VEL
LIN {X 0,Y 523.98,Z 736.996,A -85,B 0,C 180,E1 -4605.237,E2 -4605.237} C_VEL
LIN {X 0,Y 524.185,Z 725.258,A -85,B 0,C 180,E1 -4607.961,E2 -4607.961} C_VEL
LIN {X 0,Y 524.035,Z 722.124,A -85,B 0,C 180,E1 -4608.725,E2 -4608.725} C_VEL
LIN {X 0,Y 523.947,Z 722.029,A -85,B 0,C 180,E1 -4611.233,E2 -4611.233} C_VEL
LIN {X 0,Y 523.936,Z 722.036,A -85,B 0,C 180,E1 -4614.197,E2 -4614.197} C_VEL
LIN {X 0,Y 523.91,Z 722.032,A -85,B 0,C 180,E1 -4617.135,E2 -4617.135} C_VEL
LIN {X 0,Y 523.939,Z 722.03,A -85,B 0,C 180,E1 -4619.756,E2 -4619.756} C_VEL
LIN {X 0,Y 523.934,Z 722.033,A -85,B 0,C 180,E1 -4622.45,E2 -4622.45} C_VEL
LIN {X 0,Y 523.92,Z 722.032,A -85,B 0,C 180,E1 -4625.227,E2 -4625.227} C_VEL
LIN {X 0,Y 523.916,Z 722.031,A -85,B 0,C 180,E1 -4628.102,E2 -4628.102} C_VEL
LIN {X 0,Y 523.957,Z 722.026,A -85,B 0,C 180,E1 -4631.31,E2 -4631.31} C_VEL
LIN {X 0,Y 523.943,Z 722.031,A -85,B 0,C 180,E1 -4634.69,E2 -4634.69} C_VEL
LIN {X 0,Y 523.951,Z 722.011,A -85,B 0,C 180,E1 -4637.881,E2 -4637.881} C_VEL
LIN {X 0,Y 523.92,Z 722.036,A -85,B 0,C 180,E1 -4640.915,E2 -4640.915} C_VEL
LIN {X 0,Y 523.901,Z 722.032,A -85,B 0,C 180,E1 -4643.825,E2 -4643.825} C_VEL
LIN {X 0,Y 523.915,Z 722.034,A -85,B 0,C 180,E1 -4646.634,E2 -4646.634} C_VEL
LIN {X 0,Y 523.951,Z 722.03,A -85,B 0,C 180,E1 -4649.355,E2 -4649.355} C_VEL
LIN {X 0,Y 523.976,Z 722.023,A -85,B 0,C 180,E1 -4652.282,E2 -4652.282} C_VEL
LIN {X 0,Y 523.95,Z 722.024,A -85,B 0,C 180,E1 -4654.581,E2 -4654.581} C_VEL
LIN {X 0,Y 523.912,Z 722.04,A -85,B 0,C 180,E1 -4657.106,E2 -4657.106} C_VEL
LIN {X 0,Y 523.981,Z 722.022,A -85,B 0,C 180,E1 -4659.866,E2 -4659.866} C_VEL
